IF (gu8_SystemState = DRIVE_SYS AND DO_q_BatteryDischargeMain_DO = TRUE) THEN
	IF (gq_Gear_Drive_Rq = TRUE AND gq_BrakeSwitch = TRUE) AND gr_VehicleSpeed_kmph > -1 THEN
		gq_Gear_Neutral			:=	FALSE;
		gq_Gear_Drive			:=	TRUE;
		gq_Gear_DriveCrawl		:=	FALSE;
		gq_Gear_Reverse			:=	FALSE;
		gq_Gear_ReverseCrawl	:=	FALSE; (*Select Drive*)
	ELSIF (gq_Gear_Neutral_Rq = TRUE AND gq_BrakeSwitch = TRUE) AND (gr_VehicleSpeed_kmph <1 AND gr_VehicleSpeed_kmph >-1) THEN
		gq_Gear_Neutral			:=	TRUE;
		gq_Gear_Drive			:=	FALSE;
		gq_Gear_DriveCrawl		:=	FALSE;
		gq_Gear_Reverse			:=	FALSE;
		gq_Gear_ReverseCrawl	:=	FALSE; (*Select Neutral*)
	ELSIF (gq_Gear_Reverse_Rq = TRUE AND gq_BrakeSwitch = TRUE) AND gr_VehicleSpeed_kmph < 1 THEN
		gq_Gear_Neutral			:=	FALSE;
		gq_Gear_Drive			:=	FALSE;
		gq_Gear_DriveCrawl		:=	FALSE;
		gq_Gear_Reverse			:=	TRUE;
		gq_Gear_ReverseCrawl	:=	FALSE; (*Select Reverse*)
	ELSIF (DI_q_DirectionSwitch_DriveCrawl_DI = TRUE AND gq_BrakeSwitch = TRUE) THEN
		gq_Gear_Neutral			:=	FALSE;
		gq_Gear_Drive			:=	FALSE;
		gq_Gear_DriveCrawl		:=	TRUE;
		gq_Gear_Reverse			:=	FALSE;
		gq_Gear_ReverseCrawl	:=	FALSE; (*Select Drive Crawl*)
	(*ELSIF (DI_q_DirectionSwitch_ReverseCrawl_DI = TRUE AND gq_BrakeSwitch = TRUE) THEN
		gq_Gear_Neutral			:=	FALSE;
		gq_Gear_Drive			:=	FALSE;
		gq_Gear_DriveCrawl		:=	FALSE;
		gq_Gear_Reverse			:=	FALSE;
		gq_Gear_ReverseCrawl	:=	TRUE; (*Select Reverse Crawl*)*)
	END_IF
ELSIF (gu8_SystemState <> DRIVE_SYS) THEN
	gq_Gear_Neutral			:=	TRUE;
	gq_Gear_Drive			:=	FALSE;
	gq_Gear_DriveCrawl		:=	FALSE;
	gq_Gear_Reverse			:=	FALSE;
	gq_Gear_ReverseCrawl	:=	FALSE; (*Gear selection = Neutral*)
ELSE
	gq_Gear_Neutral			:=	TRUE;
	gq_Gear_Drive			:=	FALSE;
	gq_Gear_DriveCrawl		:=	FALSE;
	gq_Gear_Reverse			:=	FALSE;
	gq_Gear_ReverseCrawl	:=	FALSE; (*Neutral*)
END_IF

gq_ReverseLights	:=	gq_Gear_Reverse;

END_PROGRAM

// Application/UserCode/BMS/OrionBMS/Orion_Control
PROGRAM Orion_Control
VAR
	OrionPause_Timer	:	TON;
	hton_DisconnectionPause_Timer	:	TON;
END_VAR

(*Program to control the BMS during operation*)
(*Setting battery mode*)
IF (gu8_SystemState = DRIVE_SYS) THEN
	(*Have an initial short pause after contactors have closed before changing into discharge mode*)
	OrionPause_Timer(IN := TRUE, PT := T#20mS);
	IF (OrionPause_Timer.Q = TRUE) THEN
		(*Set discharge output*)
		DO_q_DrivetrainKL15C_DO	:=	FALSE;
		DO_q_DrivetrainKL15D_DO	:=	TRUE;
		(*Request on CAN the BMS into operational mode*)
		gu8_BMS1_MPO_1_State	:=	1;
		gu8_BMS1_MPO_2_State	:=	1; (* This does F_ALL *)
		gu8_BMS2_MPO_1_State	:=	1;
		gu8_BMS2_MPO_2_State	:=	1;
		
		
	END_IF
	hton_DisconnectionPause_Timer(IN := FALSE, PT := T#0MS);
ELSIF (gu8_SystemState = PLUGIN_SYS) THEN
	(*Have an initial short pause after contactors have closed before changing into charge mode*)
	OrionPause_Timer(IN := TRUE, PT := T#20MS);
	IF (OrionPause_Timer.Q = TRUE) THEN
		(*Set outputs for charge mode*)
		DO_q_DrivetrainKL15C_DO	:=	TRUE;
		DO_q_DrivetrainKL15D_DO	:=	FALSE;
		(*Request on CAN the BMS into operational mode*)
		gu8_BMS1_MPO_1_State	:=	0;
		gu8_BMS1_MPO_2_State	:=	0;
		gu8_BMS2_MPO_1_State	:=	0;
		gu8_BMS2_MPO_2_State	:=	0;
	END_IF
	hton_DisconnectionPause_Timer(IN := FALSE, PT := T#0MS);
ELSIF (DO_q_BatteryDischargeMain_DO = FALSE AND DO_q_Battery1ChargeMain_DO = FALSE AND DO_q_Battery2ChargeMain_DO = FALSE AND
		DO_q_BatteryDischargePrecharge_DO = FALSE AND DO_q_Battery1ChargePrecharge_DO = FALSE AND DO_q_Battery2ChargePrecharge_DO = FALSE) THEN
	(*Only perform disconnect of batteries when all contactors are opened to prevent them from damaging their own contactors Explain ??MAT *)
	hton_DisconnectionPause_Timer(IN := TRUE, PT := T#100MS);
	IF (hton_DisconnectionPause_Timer.Q = TRUE) THEN
		DO_q_DrivetrainKL15C_DO	:=	FALSE;
		DO_q_DrivetrainKL15D_DO	:=	FALSE;
		(*Request the BMS inactive*)
		gu8_BMS1_MPO_1_State	:=	0;
		gu8_BMS1_MPO_2_State	:=	0;
		gu8_BMS2_MPO_1_State	:=	0;
		gu8_BMS2_MPO_2_State	:=	0;
			
	END_IF
	OrionPause_Timer(IN := FALSE, PT := t#0ms);
END_IF
IF qq_BMS1_PB_DTC_Reset THEN
	gu8_BMS1_MPO_3_State :=1;
	ELSE gu8_BMS1_MPO_3_State :=0;
END_IF
IF qq_BMS2_PB_DTC_Reset THEN
	gu8_BMS2_MPO_3_State :=1;
	ELSE gu8_BMS2_MPO_3_State :=0;
END_IF

END_PROGRAM

// Application/UserCode/MCU/MCU_Control
PROGRAM MCU_Control
VAR
	hs8_Direction	:	SINT	:=	0;
	hton_Mileometer	:	TON;
	hq_SetInitialDistance	:	BOOL	:=	FALSE;
	hton_TorqueRqRamp	:	TON;
	hr_TorqueRampTime	:	REAL;
	hr_TorqueRampTotal	:	REAL;
	hr_MCU_TorquePreRamp	:	REAL;
	hf_TorqueRamp			:	Ramp_Linear;
	
	TORQUE_RQ_CF	:	REAL	:=	0.3; (*In case any conversion factors need to be applied to the value being sent*)
	hr_MULTIPLIER_CALC	: REAL	:= 0;
	WINDUPSPEED			: USINT := 10;
	
	hr_SpeedLimit_KP	:	REAL	:=	10;
	hr_SpeedLimit_KI	:	REAL	:=	10;
	hfb_SpeedLimit_PID	:	PID;
	hr_MaximumTorqueLimit : REAL;
	hr_TARGETMAXSPEED : REAL := 77;
	hr_IntegralCounter : ARRAY [0..49] OF REAL;
	Counter : USINT := 0;
	hr_IntegralSum : REAL := 0;
	Cycle : USINT;
END_VAR
VAR CONSTANT
	INITIALISATION	:	USINT	:=	0;
	STANDBY			:	USINT	:=	1;
	STARTUP			:	USINT	:=	2;
	TEARDOWN		:	USINT	:=	3;
	OPERATIONAL		:	USINT	:=	4;
	FAILURE			:	USINT	:=	5;
	CLOSEDOWN		:	USINT	:=	6;
	READYTOSHUTDOWN	:	USINT	:=	7;
	WAITFORCOOLING	:	USINT	:=	8;
	
	SHUTDOWN_RQ		:	USINT	:=	2;
	OPERATIONAL_RQ	:	USINT	:=	1;
	STANDBY_RQ		:	USINT	:=	0;
	
	TORQUE_MODE		:	USINT	:=	1;
	SPEED_MODE		:	USINT	:=	2;
	
	
	
	EV_MODE			:	USINT	:=	3;
	NEU_NOTORQUE	:	USINT	:=	0;

END_VAR

IF (DI_q_VehicleKL15_DI = TRUE) THEN
	hton_Mileometer(IN := TRUE, PT := T#60S);
	IF (gu16_MCU_MaxMotorSpeed_Rx = 0) THEN
		gu8_MCU_VMUPollMCU_Multiplex	:=	MAXMOTORSPEED;
	ELSIF (gu16_MCU_MaxMotorTorque_Rx = 0) THEN
		gu8_MCU_VMUPollMCU_Multiplex	:=	MAXMOTORTORQUE;
	ELSIF (hton_Mileometer.Q = TRUE) THEN
		hton_Mileometer(IN := FALSE, PT := T#0S);
		gu8_MCU_VMUPollMCU_Multiplex	:=	TOTALMOTORROTATION;
	ELSE
		gu8_MCU_VMUPollMCU_Multiplex	:=	8; (*Not applicable value so will not incorrectly request any data*)
	END_IF
END_IF

(*Must be in discharge mode and precharge complete before command out of standby (Need to set ignition at the start always)*)
IF (gu8_SystemState = DRIVE_SYS AND DOS_q_BatteryDischargeMain_DO = TRUE(* AND gr_MCU_TractionTorqueAvailable > 0*)) THEN
	IF ((gu8_MCU_State = STANDBY) AND gq_Gear_Neutral = TRUE) THEN
		gu8_MCU_OperationRequest	:=	OPERATIONAL_RQ;
		gu8_MCU_OperationalMode_Tx	:=	NEU_NOTORQUE;
	ELSIF (gu8_MCU_State = OPERATIONAL) THEN
		gu8_MCU_OperationRequest	:=	OPERATIONAL_RQ;
		gu8_MCU_OperationalMode_Tx	:=	EV_MODE;
	END_IF
ELSIF (gu8_SystemState <> DRIVE_SYS) THEN
	IF (gu8_MCU_State = OPERATIONAL AND gq_Gear_Neutral = TRUE) THEN
		gu8_MCU_OperationRequest	:=	SHUTDOWN_RQ;
		gu8_MCU_OperationalMode_Tx	:=	NEU_NOTORQUE;
	ELSIF (gu8_MCU_State = OPERATIONAL AND gq_Gear_Neutral = FALSE) THEN
		gu8_MCU_OperationRequest	:=	OPERATIONAL_RQ;
		gu8_MCU_OperationalMode_Tx	:=	NEU_NOTORQUE;
		(*Rq Neutral*)
	ELSE
		gu8_MCU_OperationRequest	:=	STANDBY_RQ;
		gu8_MCU_OperationalMode_Tx	:=	NEU_NOTORQUE;
	END_IF
ELSE
	gu8_MCU_OperationRequest	:=	STANDBY_RQ;
	gu8_MCU_OperationalMode_Tx	:=	NEU_NOTORQUE;
END_IF

(*These values should be set by the BMS*)
gu16_MCU_MaxChargeCurrent		:=	REAL_TO_UINT(gr_BMS_CCL);
gu16_MCU_MaxDischargeCurrent	:=	REAL_TO_UINT(gr_BMS_DCL);
gu16_MCU_MaxBatteryVoltage		:=	gu16_BMS_Maximum_Pack_Voltage;
gu16_MCU_MinBatteryVoltage		:=	gu16_BMS_MinimumPackVoltage;
gu8_MCU_CommandMode				:=	TORQUE_MODE;
gu8_MCU_ReferenceCommandMode	:=	TORQUE_MODE;
gr_MCU_MaxMotorSpeed_PreCF		:=	gr_MCU_MaxMotorSpeed; (*This may need to be set for safety*)

IF (gq_Gear_Drive = TRUE OR gq_Gear_DriveCrawl = TRUE) THEN
	hs8_Direction	:=	1;
	gq_MCU_SpeedCommandStatus		:=	FALSE;
	gq_MCU_TorqueCommandStatus		:=	FALSE;
ELSIF (gq_Gear_Reverse = TRUE OR gq_Gear_ReverseCrawl = TRUE) THEN
	hs8_Direction	:=	-1;
	gq_MCU_SpeedCommandStatus		:=	FALSE;
	gq_MCU_TorqueCommandStatus		:=	FALSE;
ELSE
	hs8_Direction	:=	0;
	gq_MCU_SpeedCommandStatus		:=	TRUE;
	gq_MCU_TorqueCommandStatus		:=	TRUE;
END_IF

hr_MULTIPLIER_CALC := gr_VehicleSpeed_kmph / WINDUPSPEED;
TORQUE_RQ_CF := LIMIT(1(*0.3*), hr_MULTIPLIER_CALC, 1);

Driveability();
IF (gu8_MCU_State = OPERATIONAL AND hs8_Direction <> 0 (*Not in neutral*) AND gq_ABSActive = FALSE AND gq_MCU_CutOff_LowCellV = FALSE AND gq_BodySteps = FALSE) THEN
	IF (gq_ABS_TorqueDisable = TRUE) THEN
		hton_TorqueRqRamp(IN := FALSE, PT := T#0S);
		gr_MCU_TorqueCommand_PreCF			:=	0;
	ELSIF (gq_ZeroTorqueRq = TRUE) THEN
		hton_TorqueRqRamp(IN := FALSE, PT := T#0S);
		IF (gq_RegenActive = TRUE) THEN
			gr_MCU_TorqueCommand_PreCF	:=	(*gr_MCU_MaxMotorTorque*)gr_MCU_RegenTorqueAvailable * gr_RegenSOCMultiplier * gr_RegenMultiplierRq * gr_RegenSpeedDegrading * gr_RegenIntroCF * (hs8_Direction * (-1)) * LIMIT(0, (gr_TorqueReIntro / gr_TorqueReIntroMax), 1);(**)
		ELSIF (gq_RegenActive = FALSE) THEN
			gr_MCU_TorqueCommand_PreCF			:=	gr_AccelPedal_Perc * TORQUE_RQ_CF * hs8_Direction * (*gr_MCU_MaxMotorTorque*)gr_MCU_TractionTorqueAvailable * LIMIT(0, (gr_TorqueReIntro / gr_TorqueReIntroMax), 1);
		END_IF
	ELSIF (gq_ABS_TorqueDisable = FALSE AND gq_ZeroTorqueRq = FALSE) THEN
		IF (gq_RegenActive = TRUE) THEN
			hton_TorqueRqRamp(IN := FALSE, PT := T#0S);
			gr_MCU_TorqueCommand_PreCF	:=	(*gr_MCU_MaxMotorTorque*)gr_MCU_RegenTorqueAvailable * gr_RegenSOCMultiplier * gr_RegenMultiplierRq * gr_RegenSpeedDegrading * gr_RegenIntroCF * (hs8_Direction * (-1));(**)
		ELSIF (gq_RegenActive = FALSE) THEN	
			hr_MCU_TorquePreRamp	:=	gr_AccelPedal_Perc * TORQUE_RQ_CF * hs8_Direction * (*gr_MCU_MaxMotorTorque*)gr_MCU_TractionTorqueAvailable;
			gr_MCU_TorqueCommand_PreCF	:=	hr_MCU_TorquePreRamp;
		END_IF
	END_IF
	//*DO_q_DrivetrainCoolingFan_DO		:=	TRUE;
ELSE
	gr_MCU_TorqueCommand_PreCF			:=	0 * TORQUE_RQ_CF * (*gr_MCU_MaxMotorTorque*)gr_MCU_TractionTorqueAvailable;
	//*DO_q_DrivetrainCoolingFan_DO		:=	FALSE;
	hton_TorqueRqRamp(IN := FALSE, PT := T#0S);
END_IF

IF (gu8_BMS_SOC > 10) THEN
	IF (gu8_ChassisType <> CHASSIS_IVECO) THEN
		hr_TARGETMAXSPEED := SpeedOTG;
	ELSIF (gu8_ChassisType = CHASSIS_IVECO) THEN
		hr_TARGETMAXSPEED := 55;
	END_IF
ELSE
	IF (gu8_ChassisType <> CHASSIS_IVECO) THEN
		hr_TARGETMAXSPEED := SpeedOTG1;
	ELSIF (gu8_ChassisType = CHASSIS_IVECO) THEN
		hr_TARGETMAXSPEED := 24;
	END_IF
END_IF

IF (gr_VehicleSpeed_kmph > hr_TARGETMAXSPEED) THEN
	hr_MaximumTorqueLimit := 0;
ELSE
	hr_IntegralCounter[Counter] := LIMIT(0, (hr_TARGETMAXSPEED - gr_VehicleSpeed_kmph), hr_TARGETMAXSPEED);
	IF (Counter > 49) THEN
		Counter := 0;
	ELSE
		Counter := Counter + 1;
	END_IF
	hr_IntegralSum := 0;
	FOR Cycle := 0 TO 49 DO
		hr_IntegralSum := hr_IntegralSum + hr_IntegralCounter[Cycle];
	END_FOR
	hr_MaximumTorqueLimit := MAX(((hr_TARGETMAXSPEED - gr_VehicleSpeed_kmph) * hr_SpeedLimit_KP + hr_IntegralSum * hr_SpeedLimit_KI), 0);
END_IF


gr_MCU_SpeedCommand_PreCF			:=	0;

gr_MCU_TorqueCommand_PreCF_Limited	:=	LIMIT(-3500, gr_MCU_TorqueCommand_PreCF, hr_MaximumTorqueLimit);
gr_MCU_ReferenceTorqueCommand_PreCF	:=	LIMIT(-3500, gr_MCU_TorqueCommand_PreCF, hr_MaximumTorqueLimit);
gr_MCU_ReferenceSpeedCommand_PreCF	:=	gr_MCU_SpeedCommand_PreCF;

(*Don't think I need to set these but will keep them here as a reminder and just in case they do need setting*)
gq_MCU_MaxDiscahrgeCurrentStatus	:=	FALSE;
gq_MCU_MaxBatteryVoltageStatus		:=	FALSE;
gq_MCU_MinBatteryVoltageStatus		:=	FALSE;
gq_MCU_MaxChargeCurrentStatus		:=	FALSE;

gr_VehicleSpeed_kmph	:=	f_SpeedCalc(gr_MotorSpeed_IN := gr_MCU_MotorSpeed, gu16_GearRatio_IN := gu16_GearRatio_PreCF,
										gu16_DyfRatio_IN := gu16_DyfRatio_PreCF, gu16_TireWidth_IN := gu16_TireWidth_mm,
										gu8_TireProfile_IN := gu8_TireProfile_Perc, gu16_WheelDiameter_IN := gu16_WheelDiameter_PreCF);

gr_VehicleAllTimeDistance	:=	f_DistanceCalc(gr_MotorRotation_IN := gr_MCU_TotalMotorRotation, gu16_GearRatio_IN := gu16_GearRatio_PreCF,
										gu16_DyfRatio_IN := gu16_DyfRatio_PreCF, gu16_TireWidth_IN := gu16_TireWidth_mm,
										gu8_TireProfile_IN := gu8_TireProfile_Perc, gu16_WheelDiameter_IN := gu16_WheelDiameter_PreCF);

IF (hq_SetInitialDistance = FALSE AND gr_MCU_TotalMotorRotation <> 0) THEN
	gr_VehicleInitialTripDistance	:=	gr_VehicleAllTimeDistance;
	hq_SetInitialDistance			:=	TRUE;
END_IF

gr_VehicleTripDistance	:=	gr_VehicleAllTimeDistance - gr_VehicleInitialTripDistance;

END_PROGRAM

// Application/UserCode/MCU/Driveability
PROGRAM Driveability
VAR
	hq_RegenAvailable	:	BOOL;
	hton_RegenHysteresis	:	TON;
	hr_DriveSpeed	:	REAL;
	hr_FrontSpeed	:	REAL;
	hr_LeftWheels_Speed	:	REAL;
	hr_RightWheels_Speed	:	REAL;
	hr_TractionSpdDiff	:	REAL;
	hr_StabilitySpdDiff	:	REAL;
	
	(*Traction and Stability Dennis and Iveco*)
	TRACTIONLOSS_RELSPEED	:	REAL	:=	300; (*Temporarily set high until time to configure these to the correct value*)
	STABLOSS_RELSPEED		:	REAL	:=	3; (*Temporarily set high until time to configure these to the correct value*)
	(*Bob traction and stability values*)
	TRACTIONLOSS_SPEED	:	UINT	:=	3500;
	STABLOSS_SPEED		:	UINT	:=	1000;
	
	REGEN_CUTOFF_SPEED	:	USINT	:=	5;
	REGEN_WINDDOWNABOVECUTOFF_SPEED	:	USINT	:=	25;
	hton_RegenStartTimer : TON;
	// This ideally should be set to 100ms
	htime_RegenIntro : TIME := T#100MS;
	
	// WAS 0.7 ON BRAKE
	DENNIS_ADJUSTABLE_REGEN	:	REAL	:=	0.4 (*0.4*);
	
	hr_StabilityRelativeDifference : REAL;
	hu8_StabRampSpeed	:	USINT	:=	30;
	hr_STABLOSS_HIGHSPD	:	REAL	:=	2.5;
	hr_StabIncreaseMultiplier	:	REAL	:=	3;
	hr_STABLOSS_HIGHSPD_IVECO	:	REAL	:=	1.5;
	hr_StabIncreaseMultiplier_IVECO	:	REAL	:=	2;
	
	hr_RegenTest	:	REAL	:=	1; (*Use this value in place of the constants for regen multiplier to allow changes to be made by forcing on the fly*)
	
	SecretTractionOff: BOOL;
	hton_Overspeed_Regen: TON;
END_VAR
VAR_INPUT
	Dennis_Regen_Selector: BYTE := 0;
END_VAR


(*ABS*)
IF (CAN3_Rx.Mode_Button AND CAN3_Rx.Down_Button) = TRUE THEN
	SecretTractionOff :=	TRUE;
END_IF

IF (CAN3_Rx.Mode_Button AND CAN3_Rx.Up_Button) = TRUE THEN
	SecretTractionOff := 	FALSE;
END_IF

IF (gq_ABSActive = TRUE) THEN
	gq_ABS_TorqueDisable	:=	TRUE;
ELSIF (gq_ABSActive = FALSE AND gr_AccelPedal_Perc > 0.03(*3%*)) THEN
	gq_ABS_TorqueDisable	:=	FALSE;
END_IF

IF (gq_Frosty_NoWheelSpeedSensors = TRUE) THEN
	hr_STABLOSS_HIGHSPD_IVECO	:=	10; (*Set so that Stability loss detection does not prevent drive*)
END_IF

IF (gu8_ChassisType = CHASSIS_IVECO AND gq_StabTracDisable_Rx = FALSE) THEN
	(*Traction Control*)
	gr_RearAxle_RelativeSpeed_kph	:= (gr_EBC2_KB_RearRight1RelSpd + gr_EBC2_KB_RearLeft1RelSpd) / 2;
	IF (ABS(gr_RearAxle_RelativeSpeed_kph) > TRACTIONLOSS_RELSPEED(*Change this value to be whatever the speed difference needs to be to trigger can be decimal*)) THEN
		gu8_TractionLoss	:=	1(*TRUE*);
	ELSE
		gu8_TractionLoss	:=	0(*FALSE*);
	END_IF

	(*Stability*)
	IF (gr_VehicleSpeed_kmph > hu8_StabRampSpeed) THEN
		STABLOSS_RELSPEED := hr_STABLOSS_HIGHSPD_IVECO;
	ELSE
		STABLOSS_RELSPEED := hr_STABLOSS_HIGHSPD_IVECO + ((hu8_StabRampSpeed - ABS(gr_VehicleSpeed_kmph)) * hr_StabIncreaseMultiplier_IVECO / hu8_StabRampSpeed);
	END_IF
	
	gr_LeftWheels_RelativeSpeed_kph		:=	(gr_EBC2_KB_FrontLeftRelSpd + gr_EBC2_KB_RearLeft1RelSpd) / 2;
	gr_RightWheels_RelativeSpeed_kph	:=	(gr_EBC2_KB_FrontRightRelSpd + gr_EBC2_KB_RearRight1RelSpd) / 2;
	IF (ABS(gr_LeftWheels_RelativeSpeed_kph) > STABLOSS_RELSPEED OR ABS(gr_RightWheels_RelativeSpeed_kph) > STABLOSS_RELSPEED) THEN (*Can equally use decimal numbers here if needed*)
		gu8_StabilityLoss	:=	1(*TRUE*);
	ELSE
		gu8_StabilityLoss	:=	0(*FALSE*);
	END_IF
ELSIF (gu8_ChassisType = CHASSIS_BOB OR gu8_ChassisType = CHASSIS_ESTARGLIDER) AND (gq_StabTracDisable_Rx = FALSE AND SecretTractionOff = FALSE) THEN // OR should be AND
	(*Traction Control*)
	hr_DriveSpeed	:= (gu16_Bob_RightDrive_CAN + gu16_Bob_LeftDrive_CAN) / 2;
	hr_FrontSpeed	:= (gu16_Bob_RightFront_CAN + gu16_Bob_LeftFront_CAN) / 2;
	hr_TractionSpdDiff	:=	ABS(hr_DriveSpeed - hr_FrontSpeed);
	IF (hr_TractionSpdDiff > TRACTIONLOSS_SPEED(*Change this value to be whatever the speed difference needs to be to trigger can be decimal*)) THEN
		gu8_TractionLoss	:=	1(*TRUE*);
	ELSE
		gu8_TractionLoss	:=	0(*FALSE*);
	END_IF
	(*Stability*)
	hr_LeftWheels_Speed		:=	(gu16_Bob_LeftFront_CAN + gu16_Bob_LeftDrive_CAN) / 2;
	hr_RightWheels_Speed	:=	(gu16_Bob_RightFront_CAN + gu16_Bob_RightDrive_CAN) / 2;
	hr_StabilitySpdDiff		:=	ABS(hr_LeftWheels_Speed - hr_RightWheels_Speed);
	IF (hr_StabilitySpdDiff > STABLOSS_SPEED) THEN (*Can equally use decimal numbers here if needed*)
		gu8_StabilityLoss	:=	1(*TRUE*);
	ELSE
		gu8_StabilityLoss	:=	0(*FALSE*);
	END_IF
ELSIF (gu8_ChassisType = CHASSIS_DENNIS AND (gq_StabTracDisable_Rx = FALSE AND SecretTractionOFF = FALSE)) THEN
	(*Traction Control*)
	(*gr_RearAxle_RelativeSpeed_kph	:= (gr_EBC2_KB_RearRight1RelSpd + gr_EBC2_KB_RearLeft1RelSpd) / 2;
	IF (ABS(gr_RearAxle_RelativeSpeed_kph) > TRACTIONLOSS_RELSPEED(*Change this value to be whatever the speed difference needs to be to trigger can be decimal*)) THEN
		gu8_TractionLoss	:=	1(*TRUE*);
	ELSE
		gu8_TractionLoss	:=	0(*FALSE*);
	END_IF*)
	(*Stability*)
	IF (gr_VehicleSpeed_kmph > hu8_StabRampSpeed) THEN
		STABLOSS_RELSPEED := hr_STABLOSS_HIGHSPD;
	ELSE
		STABLOSS_RELSPEED := hr_STABLOSS_HIGHSPD + ((hu8_StabRampSpeed - ABS(gr_VehicleSpeed_kmph)) * hr_StabIncreaseMultiplier / hu8_StabRampSpeed);
	END_IF
	
	gr_LeftWheels_RelativeSpeed_kph		:=	(gr_EBC2_KB_FrontLeftRelSpd + gr_EBC2_KB_RearLeft1RelSpd) / 2;
	gr_RightWheels_RelativeSpeed_kph	:=	(gr_EBC2_KB_FrontRightRelSpd + gr_EBC2_KB_RearRight1RelSpd) / 2;
	hr_StabilityRelativeDifference	:=	ABS(gr_LeftWheels_RelativeSpeed_kph - gr_RightWheels_RelativeSpeed_kph);
	IF (*(ABS(gr_LeftWheels_RelativeSpeed_kph) > STABLOSS_RELSPEED OR ABS(gr_RightWheels_RelativeSpeed_kph) > STABLOSS_RELSPEED)*)
		(hr_StabilityRelativeDifference > STABLOSS_RELSPEED) THEN (*Can equally use decimal numbers here if needed*)
		gu8_StabilityLoss	:=	1(*TRUE*);
	ELSE
		gu8_StabilityLoss	:=	0(*FALSE*);
	END_IF
	gu8_TractionLoss	:=	gu8_EBC1_ASREngineControlActive;
	(*gu8_StabilityLoss	:=	gu8_EBC1_ASRBrakeControlActive;*)
ELSIF (gq_StabTracDisable_Rx = TRUE) THEN
	gu8_TractionLoss	:=	0(*FALSE*);
	gu8_StabilityLoss	:=	0(*FALSE*);
END_IF


(*Zero torque and Recovery*)
IF (gu8_TractionLoss = 1 OR gu8_StabilityLoss = 1 (* REAMED by IAIN 121021 OR Sevcon2_Control.NO_OIL*)) THEN
	gq_ZeroTorqueRq	:=	TRUE;
	gton_TorqueReIntro_Timer(IN := FALSE, PT := T#0MS);
ELSE
	gton_TorqueReIntro_Timer(IN := TRUE, PT := T#2000MS);
END_IF
IF (gton_TorqueReIntro_Timer.Q = TRUE) THEN
	gq_ZeroTorqueRq	:=	FALSE;
END_IF
gr_TorqueReIntro	:=	TIME_TO_REAL(gton_TorqueReIntro_Timer.ET);
gr_TorqueReIntroMax	:=	TIME_TO_REAL(T#2000MS);

(*Regen*)
(*Selectable regen setting needed*)
IF (gu8_BMS_SOC < 90) THEN
	gr_RegenSOCMultiplier	:=	1;
ELSIF (gu8_BMS_SOC >= 90 AND gu8_BMS_SOC < 95) THEN
	gr_RegenSOCMultiplier	:=	0.5;
ELSE
	gr_RegenSOCMultiplier	:=	0;
END_IF


IF (gr_VehicleSpeed_kmph > REGEN_CUTOFF_SPEED) THEN
	hton_RegenHysteresis(IN := TRUE, PT := T#1000MS); // bring down to T#1s? Was t#5s
ELSE
	hton_RegenHysteresis(IN := FALSE, PT := T#0S);
END_IF
hq_RegenAvailable	:=	hton_RegenHysteresis.Q;

hton_Overspeed_Regen (IN:= gr_VehicleSpeed_kmph > 55, PT:= T#5S);
IF ((gr_AccelPedal_Perc < 0.01 OR (gr_VehicleSpeed_kmph > 55 AND hton_Overspeed_Regen.Q)) AND hq_RegenAvailable = TRUE) THEN //OR gr_VehicleSpeed_kmph > 56 added
	gq_RegenActive	:=	TRUE;
	gr_RegenSpeedDegrading	:=	LIMIT(0, (gr_VehicleSpeed_kmph - REGEN_CUTOFF_SPEED), REGEN_WINDDOWNABOVECUTOFF_SPEED) / REGEN_WINDDOWNABOVECUTOFF_SPEED;
	IF gr_VehicleSpeed_kmph > 55 THEN
	DENNIS_ADJUSTABLE_REGEN := 1.2;
	END_IF
//////////////	

//DENNIS with BRAKE
	IF (gu8_ChassisType = CHASSIS_DENNIS AND gq_BrakeSwitch = TRUE) THEN
		DENNIS_ADJUSTABLE_REGEN := 1.2;
		gr_RegenMultiplierRq	:=	DENNIS_ADJUSTABLE_REGEN;
		hton_RegenStartTimer(IN := TRUE, PT := htime_RegenIntro);
		gr_RegenIntroCF := LIMIT(0, (TIME_TO_REAL(hton_RegenStartTimer.ET) / TIME_TO_REAL(hton_RegenStartTimer.PT)), 1);
	END_IF
//DENNIS without BRAKE	
	IF (gu8_ChassisType = CHASSIS_DENNIS AND gq_BrakeSwitch = FALSE) THEN
		gr_RegenMultiplierRq	:=	DENNIS_ADJUSTABLE_REGEN(*40%*);
		hton_RegenStartTimer(IN := TRUE, PT := htime_RegenIntro);
		gr_RegenIntroCF := LIMIT(0, (TIME_TO_REAL(hton_RegenStartTimer.ET) / TIME_TO_REAL(hton_RegenStartTimer.PT)), 1);
		
		IF Dennis_Regen.RegenCounterValue = 0 THEN 
			DENNIS_ADJUSTABLE_REGEN := 0;
		END_IF
		IF Dennis_Regen.RegenCounterValue = 1 THEN
			DENNIS_ADJUSTABLE_REGEN := 0.6;
		END_IF
		IF Dennis_Regen.RegenCounterValue = 2 THEN
			DENNIS_ADJUSTABLE_REGEN := 0.8;
		END_IF
		IF Dennis_Regen.RegenCounterValue = 3 THEN
			DENNIS_ADJUSTABLE_REGEN := 1;
		END_IF
		IF Dennis_Regen.RegenCounterValue = 4 THEN
			DENNIS_ADJUSTABLE_REGEN := 1.2;
		END_IF	
//////////////		

ELSIF (gq_BrakeSwitch = TRUE AND gu8_ChassisType <> CHASSIS_DENNIS) THEN
		IF (gu8_RegenSelector = 0) THEN
			gr_RegenMultiplierRq	:=	0.7(*40%*);
			hton_RegenStartTimer(IN := TRUE, PT := htime_RegenIntro);
			gr_RegenIntroCF := LIMIT(0, (TIME_TO_REAL(hton_RegenStartTimer.ET) / TIME_TO_REAL(hton_RegenStartTimer.PT)), 1);
		ELSIF (gu8_RegenSelector = 1) THEN
			gr_RegenMultiplierRq	:=	0.7(*40%*);
			hton_RegenStartTimer(IN := TRUE, PT := htime_RegenIntro);
			gr_RegenIntroCF := LIMIT(0, (TIME_TO_REAL(hton_RegenStartTimer.ET) / TIME_TO_REAL(hton_RegenStartTimer.PT)), 1);
		ELSIF (gu8_RegenSelector = 2) THEN
			gr_RegenMultiplierRq	:=	0.7(*60%*);
			hton_RegenStartTimer(IN := TRUE, PT := htime_RegenIntro);
			gr_RegenIntroCF := LIMIT(0, (TIME_TO_REAL(hton_RegenStartTimer.ET) / TIME_TO_REAL(hton_RegenStartTimer.PT)), 1);
		END_IF
	ELSIF (gq_BrakeSwitch = FALSE AND gu8_ChassisType <> CHASSIS_DENNIS) THEN
		IF (gu8_RegenSelector = 0) THEN
			gr_RegenMultiplierRq	:=	0(*0%*);
			hton_RegenStartTimer(IN := FALSE, PT := T#0MS);
			gr_RegenIntroCF := 0;
		ELSIF (gu8_RegenSelector = 1) THEN
			gr_RegenMultiplierRq	:=	0.6(*0.4(*40%*)*);
			hton_RegenStartTimer(IN := TRUE, PT := htime_RegenIntro);
			gr_RegenIntroCF := LIMIT(0, (TIME_TO_REAL(hton_RegenStartTimer.ET) / TIME_TO_REAL(hton_RegenStartTimer.PT)), 1);
		ELSIF (gu8_RegenSelector = 2) THEN
			gr_RegenMultiplierRq	:=	1(*0.6(*60%*)*);
			hton_RegenStartTimer(IN := TRUE, PT := htime_RegenIntro);
			gr_RegenIntroCF := LIMIT(0, (TIME_TO_REAL(hton_RegenStartTimer.ET) / TIME_TO_REAL(hton_RegenStartTimer.PT)), 1);
		END_IF
	END_IF
ELSE
	gq_RegenActive	:=	FALSE;
	gr_RegenMultiplierRq	:=	0;
	hton_RegenStartTimer(IN := FALSE, PT := T#0MS);
	gr_RegenIntroCF := 0;
END_IF
(*Also need battery SOC as multiplier <90 x1, 90<X<95 x0.5, >95 x0*)





(*Creep / Hill hold*)

END_PROGRAM

// Application/UserCode/Sevcon_Compressor/Sevcon2_Control
PROGRAM Sevcon2_Control
VAR
	hton_WindUpTorque_Timer	:	TON;
	hton_AirPressureExceeded_Timer	:	TON;
	htof_AirpressureRelief_Timer	:	TOF;
	hq_AirCompressorEnable	:	BOOL;
	hton_AirPressureDelayTimer	:	TON;
	
	hq_AirReliefValveOff : BOOL;
	
	
	hton_Compressor_Oil_Switch: TON;
	Low_Oil: BOOL;
	NO_OIL: BOOL;
	Oil_Temp_Setpoint: BYTE := 30;
	Oil_Level_Warning: BOOL;
	Compressor_Temp_Warning: BOOL;
	Comp_Motor_Temp_SP_Warning: INT := 100; //LM change from 55
	Comp_Motor_Temp_SP_Fault: INT := 120;  //LM change from 65
	Compressor_Temp_Fault: BOOL;
	Air_Temp_SP_Warning: INT := 100;
	Air_Temp_SP_Fault: INT := 120;
	Air_Temp_Warning: BOOL;
	Air_Temp_Fault: BOOL;
	BlowOffTime: TIME := T#1S;
	AirSuspensionPressure: REAL := 14.9;
	APRTimerET: TIME := t#0.5s;
	AirPressureReliefTime: TIME := t#1s;
	hton_Compressor_Run_Timer: TON;
	CRT_Trigger: BOOL;
	CRT_Time: TIME := t#60s;
	Run_on_Brake_Pressure: REAL := 9.5;
	CRT_Timer: TON;
	PVCT: TON;
	PVCT_Time: TIME := T#60s;
END_VAR
VAR CONSTANT
	(*Statuswords*)
	NOTREADY_STAT				:	USINT	:=	1;
	SHUTDOWN_STAT				:	USINT	:=	2;
	PRECHARGE_STAT				:	USINT	:=	4;
	ENERGISED_STAT				:	USINT	:=	7;
	ENABLED_STAT				:	USINT	:=	8;
	FAULTREACTIONACTIVE_STAT	:	USINT	:=	11;
	FAULTOFF_STAT				:	USINT	:=	13;
	ACTIVESHORT_STAT			:	USINT	:=	14;
	(*Commandwords*)
	NOCOMMAND_COMM		:	USINT	:=	0;
	ENERGISE_COMM		:	USINT	:=	3;
	ENABLED_COMM		:	USINT	:=	5;
	SHUTDOWN_COMM		:	USINT	:=	6;
	FAULTRESET_COMM		:	USINT	:=	9;
	ACTIVESHORT_COMM	:	USINT	:=	10;
	
	(*LOWAIRPRESSURE		:	REAL	:=	7.2; (*Need to define what the low air pressure value that is reported is*)
	HIGHAIRPRESSURE		:	REAL	:=	10;
	LOWAIRPRESSURE_BOB		:	REAL	:=	10; (*Need to define what the low air pressure value that is reported is*)
	HIGHAIRPRESSURE_BOB		:	REAL	:=	12.2(*Glider*) (*12.3 for Bob*);*)
	
	
	TORQUE_RQ			:	USINT	:=	200;
	REVERSE_SPD_LIMIT	:	INT		:=	-500;
	MAX_DISCHARGE		:	USINT	:=	50;
	MAX_CHARGE			:	SINT	:=	-50;
	TRACTION_LIMIT		:	USINT	:=	100;
END_VAR


(**)
(*Check for Comms fault*)
IF (gu8_SystemState = DRIVE_SYS AND DOS_q_BatteryDischargeMain_DO = TRUE) THEN
	IF (gu8_Sevcon2_InverterStatus = FAULTOFF_STAT OR gu8_Sevcon2_InverterStatus = ACTIVESHORT_STAT) THEN
		gu16_Sevcon2_Controlword	:=	FAULTRESET_COMM;
	ELSIF (gu8_Sevcon2_InverterStatus = NOTREADY_STAT OR gu8_Sevcon2_InverterStatus = SHUTDOWN_STAT) THEN
		gu16_Sevcon2_Controlword	:=	ENERGISE_COMM;
	ELSIF (gu8_Sevcon2_InverterStatus = PRECHARGE_STAT) THEN
		gu16_Sevcon2_Controlword	:=	ENERGISE_COMM;
	ELSIF (gu8_Sevcon2_InverterStatus = ENERGISED_STAT) THEN
		gu16_Sevcon2_Controlword	:=	ENABLED_COMM;
	ELSIF (gu8_Sevcon2_InverterStatus = ENABLED_STAT) THEN
		gu16_Sevcon2_Controlword	:=	ENABLED_COMM; (*Need a way to switch off*)
	ELSE
		gu16_Sevcon2_Controlword	:=	NOCOMMAND_COMM;
	END_IF
ELSE
	gu16_Sevcon2_Controlword	:=	SHUTDOWN_COMM;
END_IF

CRT_Timer (IN:= NOT hq_AirCompressorEnable, PT := CRT_Time); //Active when compressor hasnt run
hton_AirPressureDelayTimer(IN := TRUE, PT := T#2000MS);
PVCT (IN :=  hq_AirCompressorEnable, PT := PVCT_Time); // Compressor run-on timer

IF (hton_AirPressureDelayTimer.Q = TRUE) THEN
	IF (gq_APU_Installed = FALSE) THEN
		IF 	//(gr_J1939_AirSuspensionSupplyPress > gr_HighAirPressure_CutOff OR
			(gr_J1939_ServiceBrakeAirPressCircuit1 > gr_HighAirPressure_CutOff OR
			gr_J1939_ServiceBrakeAirPressCircuit2 > gr_HighAirPressure_CutOff) THEN
			hton_AirPressureExceeded_Timer(IN := TRUE, PT := BlowOffTime);
		ELSE
			hton_AirPressureExceeded_Timer(IN := FALSE, PT := T#1S); //changed from 0 to 2s to increase hysteresis
		END_IF
		IF (gu8_SystemState = DRIVE_SYS AND DOS_q_BatteryDischargeMain_DO = TRUE AND
			NO_OIL = FALSE AND Compressor_Temp_Fault = FALSE) (*AND gq_Bob_AirCompressorStatus_CAN = TRUE)*) THEN
			IF  (gr_VehicleSpeed_kmph > 5 AND (gr_J1939_ServiceBrakeAirPressCircuit1 < Run_on_Brake_Pressure)) OR // added to increase duty cycle
				
				//(PVCT.Q = FALSE AND CRT_Timer.Q = TRUE AND gr_VehicleSpeed_kmph > 2) OR // runs compressor for a time period
				
				((gr_J1939_AirSuspensionSupplyPress < gr_LowAirPressure_Intro OR
				gr_J1939_ServiceBrakeAirPressCircuit1 < gr_LowAirPressure_Intro OR
				gr_J1939_ServiceBrakeAirPressCircuit2 < gr_LowAirPressure_Intro) AND
				gq_DriveMode_CutOff_LowCellV = FALSE) THEN
					gu16_Sevcon2_SpeedLimitForward	:=	2600; (*Controlling the speed through the limits*)
					hq_AirCompressorEnable	:=	TRUE;
			ELSIF ((hton_AirPressureExceeded_Timer.Q = TRUE) OR (gr_VehicleSpeed_kmph > 5 AND (gr_J1939_ServiceBrakeAirPressCircuit1 > Run_on_Brake_Pressure))) THEN
				//(PVCT.Q = TRUE AND CRT_Timer.Q = FALSE AND gr_VehicleSpeed_kmph < 2) THEN // added to increase duty cycle
				gu16_Sevcon2_SpeedLimitForward	:=	0;
				hq_AirCompressorEnable	:=	FALSE;
			END_IF
		ELSE
			gu16_Sevcon2_SpeedLimitForward	:=	0;
			hq_AirCompressorEnable	:=	FALSE;
		END_IF
	
	(*For Bob possibly use
	(*gq_Bob_AirCompressorStatus_CAN = FALSE AND hq_AirReliefValveOff = TRUE)*)
	See below for how it was implemented*)
		
	(*This is needed for when the compressor is being controlled by the APU not yet*)
	ELSE
		(*IF (gr_J1939_AirSuspensionSupplyPress > HIGHAIRPRESSURE_BOB AND
			(gr_J1939_ServiceBrakeAirPressCircuit1 > HIGHAIRPRESSURE_BOB AND
			gr_J1939_ServiceBrakeAirPressCircuit2 > HIGHAIRPRESSURE_BOB))				
			(*gq_Bob_AirCompressorStatus_CAN = FALSE AND hq_AirReliefValveOff = TRUE)*) THEN
			hton_AirPressureExceeded_Timer(IN := TRUE, PT := T#1000MS);
		ELSE
			hton_AirPressureExceeded_Timer(IN := FALSE, PT := T#0MS);
		END_IF*)
		IF (gu8_SystemState = DRIVE_SYS AND DOS_q_BatteryDischargeMain_DO = TRUE AND
			NO_OIL = FALSE AND Compressor_Temp_Fault = FALSE AND gq_Bob_AirCompressorStatus_CAN = TRUE) THEN
			IF (gq_Merc_AirComp_Rq = TRUE AND gq_DriveMode_CutOff_LowCellV = FALSE) OR (htof_AirpressureRelief_Timer.ET > APRTimerET) THEN
					gu16_Sevcon2_SpeedLimitForward	:=	2600; (*Controlling the speed through the limits*)
					hq_AirCompressorEnable	:=	TRUE;
			ELSE(*ELSIF (hton_AirPressureExceeded_Timer.Q = TRUE) THEN*)
				gu16_Sevcon2_SpeedLimitForward	:=	0;
				hq_AirCompressorEnable	:=	FALSE;
			END_IF
		ELSE
			gu16_Sevcon2_SpeedLimitForward	:=	0;
			hq_AirCompressorEnable	:=	FALSE;
		END_IF
		(*hq_AirReliefValveOff := gq_Bob_AirCompressorStatus_CAN;*)
	END_IF
END_IF
(*gq_Merc_AirComp_Enabled	:=	hq_AirCompressorEnable;*)


htof_AirpressureRelief_Timer(IN := gq_Merc_AirComp_Rq, PT := AirPressureReliefTime);
IF htof_AirpressureRelief_Timer.Q THEN
	hq_AirCompressorEnable	:=	TRUE;
	(*(hq_AirCompressorEnable = TRUE AND gs16_Sevcon2_SpeedMeasured < 1000 )) THEN*)
	gu16_Sevcon2_SpeedLimitForward	:=	2600; (*Controlling the speed through the limits*)
	hq_AirCompressorEnable	:=	TRUE;
ELSE
		;
END_IF


(*All these are constants to be sent out to the Sevcon unit and do not need changing during operation*)
IF (gu8_Sevcon2_InverterStatus = ENABLED_STAT) THEN
	hton_WindUpTorque_Timer(IN := TRUE, PT := T#5000MS);
	gr_Sevcon2_TorqueRq						:=	TORQUE_RQ * (TIME_TO_REAL(hton_WindUpTorque_Timer.ET) / 5000);
ELSE
	hton_WindUpTorque_Timer(IN := FALSE, PT := T#0MS);
	gr_Sevcon2_TorqueRq						:=	0;
END_IF
	
gr_Sevcon2_DCLink_VoltageTarget			:=	0; (*Not needed as not being used as a generator*)
gs16_Sevcon2_SpeedLimitReverse			:=	REVERSE_SPD_LIMIT;
gu16_Sevcon2_DCLink_ImaxDischarge		:=	MAX_DISCHARGE;
gs16_Sevcon2_DCLink_ImaxRecharge		:=	MAX_CHARGE;
gr_Sevcon2_TorqueTractionLimit			:=	TRACTION_LIMIT;
gr_Sevcon2_TorqueRegenLimit				:=	0;

gu8_Sevcon2_CSCommand1					:=	0;
gu8_Sevcon2_CSCommand2					:=	0;
gu8_Sevcon2_CSCurrentLimits				:=	0;
(*Counters to run every cycle and increment so the Sevcons know the VMU is still running*)
IF (gu8_Sevcon2_SEQCommand1 < 255) THEN
	gu8_Sevcon2_SEQCommand1			:=	gu8_Sevcon2_SEQCommand1 + 1;
ELSE
	gu8_Sevcon2_SEQCommand1			:=	0;
END_IF
IF (gu8_Sevcon2_SEQCommand2 < 255) THEN
	gu8_Sevcon2_SEQCommand2			:=	gu8_Sevcon2_SEQCommand2 + 1;
ELSE
	gu8_Sevcon2_SEQCommand2			:=	0;
END_IF
IF (gu8_Sevcon2_SEQCurrentLimits < 255) THEN
	gu8_Sevcon2_SEQCurrentLimits	:=	gu8_Sevcon2_SEQCurrentLimits + 1;
ELSE
	gu8_Sevcon2_SEQCurrentLimits	:=	0;
END_IF
(**************************************************************)
hton_Compressor_Oil_Switch(IN:= Low_Oil, PT:= T#2M);
IF Sevcon2_Rx.Compressor_Oil_Switch < 1 (*Rimmed AND gs16_Sevcon2_MotorTemp < Oil_Temp_Setpoint *) AND  gs16_Sevcon2_SpeedMeasured <2000 THEN
	Low_Oil := FALSE; (*changed due to poor switching*)
ELSE
	Low_Oil := FALSE;
END_IF

IF hton_Compressor_Oil_Switch.Q THEN
	NO_OIL := FALSE;
ELSE
	NO_OIL := FALSE;
END_IF

IF hton_Compressor_Oil_Switch.ET > T#30S THEN
	Oil_Level_Warning := TRUE;
ELSE
	Oil_Level_Warning := FALSE;
END_IF

IF gs16_Sevcon2_MotorTemp > Comp_Motor_Temp_SP_Warning THEN
	Compressor_Temp_Warning	:= TRUE;
ELSE
	Compressor_Temp_Warning	:= FALSE;
END_IF

IF	gs16_Sevcon2_MotorTemp > Comp_Motor_Temp_SP_Fault THEN
	Compressor_Temp_Fault := TRUE;
ELSE
	Compressor_Temp_fault := FALSE;
END_IF

IF	Sevcon2_Rx.Compressor_Temperature > Air_Temp_SP_Warning THEN
	Air_Temp_Warning := TRUE;
ELSE
	Air_Temp_Warning := FALSE;
END_IF

IF	Sevcon2_Rx.Compressor_Temperature > Air_Temp_SP_Fault THEN
	Air_Temp_Fault := TRUE;
ELSE
	Air_Temp_Fault := FALSE;
END_IF

END_PROGRAM

// Application/UserCode/MCU/f_SpeedCalc
FUNCTION f_SpeedCalc : REAL
VAR_INPUT
	gr_MotorSpeed_IN		:	REAL;
	gu16_GearRatio_IN		:	UINT;
	gu16_DyfRatio_IN		:	UINT;
	gu16_TireWidth_IN		:	UINT;
	gu8_TireProfile_IN		:	USINT;
	gu16_WheelDiameter_IN	:	UINT;
END_VAR
VAR
	hr_SidewallWidth_m	:	REAL;
	hr_TotalWheelDiameter_m	:	REAL;
	hr_WheelCircumfrence_km	:	REAL;
	hr_RevsPerKm			:	REAL;
	
	hr_GearRatio				:	REAL;
	hr_DyfRatio					:	REAL;
	hr_WheelDiameter_inch		:	REAL;
	hr_WheelDiameter_m			:	REAL;
END_VAR
VAR CONSTANT
	PI	:	REAL	:=	3.14159;
	INCH_TO_METER_CF	:	REAL	:=	0.0254;
	MILLI_TO_METER		:	UINT	:=	1000;
END_VAR


hr_GearRatio				:=	gu16_GearRatio_IN / 1000;
hr_DyfRatio					:=	gu16_DyfRatio_IN / 1000;
hr_WheelDiameter_inch		:=	gu16_WheelDiameter_IN / 10;

hr_WheelDiameter_m			:=	hr_WheelDiameter_inch * INCH_TO_METER_CF;
hr_SidewallWidth_m			:=	gu16_TireWidth_mm * (gu8_TireProfile_Perc / 100) / MILLI_TO_METER;
hr_TotalWheelDiameter_m		:=	hr_WheelDiameter_m + hr_SidewallWidth_m;

hr_WheelCircumfrence_km		:=	(hr_TotalWheelDiameter_m * PI) / 1000;
hr_RevsPerKm				:=	1 / hr_WheelCircumfrence_km;

f_SpeedCalc	:=	gr_MotorSpeed_IN / hr_GearRatio / hr_DyfRatio / hr_RevsPerKm * 60;

END_FUNCTION

// Application/UserCode/MCU/f_DistanceCalc
FUNCTION f_DistanceCalc : REAL
VAR_INPUT
	gr_MotorRotation_IN		:	REAL;
	gu16_GearRatio_IN		:	UINT;
	gu16_DyfRatio_IN		:	UINT;
	gu16_TireWidth_IN		:	UINT;
	gu8_TireProfile_IN		:	USINT;
	gu16_WheelDiameter_IN	:	UINT;
END_VAR
VAR
	hr_SidewallWidth_m	:	REAL;
	hr_TotalWheelDiameter_m	:	REAL;
	hr_WheelCircumfrence_km	:	REAL;
	hr_RevsPerKm			:	REAL;
	
	hr_GearRatio				:	REAL;
	hr_DyfRatio					:	REAL;
	hr_WheelDiameter_inch		:	REAL;
	hr_WheelDiameter_m			:	REAL;
END_VAR
VAR CONSTANT
	PI	:	REAL	:=	3.14159;
	INCH_TO_METER_CF	:	REAL	:=	0.0254;
	MILLI_TO_METER		:	UINT	:=	1000;
END_VAR


hr_GearRatio				:=	gu16_GearRatio_IN / 1000;
hr_DyfRatio					:=	gu16_DyfRatio_IN / 1000;
hr_WheelDiameter_inch		:=	gu16_WheelDiameter_IN / 10;

hr_WheelDiameter_m			:=	hr_WheelDiameter_inch * INCH_TO_METER_CF;
hr_SidewallWidth_m			:=	gu16_TireWidth_mm * (gu8_TireProfile_Perc / 100) / MILLI_TO_METER;
hr_TotalWheelDiameter_m		:=	hr_WheelDiameter_m + hr_SidewallWidth_m;

hr_WheelCircumfrence_km		:=	(hr_TotalWheelDiameter_m * PI) / 1000;
hr_RevsPerKm				:=	1 / hr_WheelCircumfrence_km;

f_DistanceCalc	:=	gr_MotorRotation_IN / hr_GearRatio / hr_DyfRatio / hr_RevsPerKm;

END_FUNCTION

// Application/UserCode/BELDCDC/BELDCDC_Control
PROGRAM BELDCDC_Control
VAR
	hton_DelayTimer	:	TON;
END_VAR

(*Setting the digital outputs to the DCDC*)

IF (DOS_q_BatteryDischargeMain_DO = TRUE AND gu8_SystemState = DRIVE_SYS) THEN
	(*Once the main contactor is connected wait 5 seconds then set the ouputs high*)
	hton_DelayTimer(IN := TRUE, PT := T#5S);
	DO_q_DrivetrainDCDCInhibit_DO	:=	hton_DelayTimer.Q;
	DO_q_DashboardDCDCStatus_DO		:=	hton_DelayTimer.Q;
ELSIF (DO_q_Battery1ChargeMain_DO = TRUE OR DO_q_Battery2ChargeMain_DO = TRUE) THEN
	(*Switch off outputs when in charge*)
	hton_DelayTimer(IN := FALSE, PT := T#0S);
	DO_q_DrivetrainDCDCInhibit_DO	:=	FALSE;
	DO_q_DashboardDCDCStatus_DO		:=	FALSE;
	(*This is included for future so that the DCDC can be brought in during charge but is not possible with current electrical setup*)
ELSE
	(*Any other state switch outputs off*)
	hton_DelayTimer(IN := FALSE, PT := T#0S);
	DO_q_DrivetrainDCDCInhibit_DO	:=	FALSE;
	DO_q_DashboardDCDCStatus_DO		:=	FALSE;
END_IF

END_PROGRAM

// Application/UserCode/Sevcon_PSP/Sevcon_Steer_Control
PROGRAM Sevcon_Steer_Control
VAR
	hton_WindUpTorque_Timer	:	TON;
	hq_PowerSteering_Enable	:	BOOL;
	hton_HandbrakeOffTimer	:	TON;
	hr_SteeringSpeed		:	REAL;
	hton_PowerSteeringOff	:	TON;
	Steering_Speed_Setpoint: INT := 2200; //changed from 2000
END_VAR
VAR CONSTANT
	(*Statuswords*)
	NOTREADY_STAT				:	USINT	:=	1;
	SHUTDOWN_STAT				:	USINT	:=	2;
	PRECHARGE_STAT				:	USINT	:=	4;
	ENERGISED_STAT				:	USINT	:=	7;
	ENABLED_STAT				:	USINT	:=	8;
	FAULTREACTIONACTIVE_STAT	:	USINT	:=	11;
	FAULTOFF_STAT				:	USINT	:=	13;
	ACTIVESHORT_STAT			:	USINT	:=	14;
	(*Commandwords*)
	NOCOMMAND_COMM		:	USINT	:=	0;
	ENERGISE_COMM		:	USINT	:=	3;
	ENABLED_COMM		:	USINT	:=	5;
	SHUTDOWN_COMM		:	USINT	:=	6;
	FAULTRESET_COMM		:	USINT	:=	9;
	ACTIVESHORT_COMM	:	USINT	:=	10;
	
	TORQUE_RQ			:	USINT	:=	200;
	REVERSE_SPD_LIMIT	:	INT		:=	-500;
	MAX_DISCHARGE		:	USINT	:=	50;
	MAX_CHARGE			:	SINT	:=	-50;
	TRACTION_LIMIT		:	USINT	:=	100;
	
	CANBUS_OFF			:	INT	:=	21256;
END_VAR


(**)
(*Check for Comms fault*)
IF (gu8_SystemState = DRIVE_SYS AND DOS_q_BatteryDischargeMain_DO = TRUE) THEN
	DO_q_DrievtrainPowerSteering_DO	:=	TRUE;
	IF (gu8_Sevcon1_InverterStatus = FAULTOFF_STAT OR gu8_Sevcon1_InverterStatus = ACTIVESHORT_STAT) THEN
		gu16_Sevcon1_Controlword	:=	FAULTRESET_COMM;
	ELSIF (gu8_Sevcon1_InverterStatus = NOTREADY_STAT OR gu8_Sevcon1_InverterStatus = SHUTDOWN_STAT) THEN
		gu16_Sevcon1_Controlword	:=	ENERGISE_COMM;
	ELSIF (gu8_Sevcon1_InverterStatus = PRECHARGE_STAT) THEN
		gu16_Sevcon1_Controlword	:=	ENERGISE_COMM;
	ELSIF (gu8_Sevcon1_InverterStatus = ENERGISED_STAT) THEN
		gu16_Sevcon1_Controlword	:=	ENABLED_COMM;
	ELSIF (gu8_Sevcon1_InverterStatus = ENABLED_STAT) THEN
		gu16_Sevcon1_Controlword	:=	ENABLED_COMM;
	ELSE
		gu16_Sevcon1_Controlword	:=	NOCOMMAND_COMM;
	END_IF
ELSE
	DO_q_DrievtrainPowerSteering_DO	:=	FALSE;
	gu16_Sevcon1_Controlword	:=	SHUTDOWN_COMM;
END_IF

hton_HandbrakeOffTimer(IN := HMI_Rx.gq_Dennis_Handbrake, PT := T#10MS); //Time changed from 30s to 10ms

(*This could be changed to link to the current speed of the vehicle in which case the different gear ratios and wheel diameter will be needed here to calculate*)
IF ((HMI_Rx.gq_Dennis_Handbrake = FALSE OR NOT gq_Gear_Neutral) AND gu8_SystemState = DRIVE_SYS) THEN //TEST FIRST THEN REMOVE THIS COMMENT OR NOT gq_Gear_Neutral
	hq_PowerSteering_Enable	:=	TRUE;
	hr_SteeringSpeed		:=	MAX(REAL_TO_INT(Steering_Speed_Setpoint - (ABS(gr_VehicleSpeed_kmph) * 10)), 0) (*Ensure the speed limit is never set negative*);
	gu16_Sevcon1_SpeedLimitForward	:=	REAL_TO_UINT(LIMIT(200, hr_SteeringSpeed, Steering_Speed_Setpoint)); (*Controlling the speed through the limits*)
	hton_PowerSteeringOff(IN := FALSE, PT := T#0S);
ELSIF ((hton_HandbrakeOffTimer.Q = TRUE AND ABS(gr_VehicleSpeed_kmph) < 3) AND gu8_SystemState = DRIVE_SYS) THEN //AND before DRIVE_SYS changed from OR
	hq_PowerSteering_Enable	:=	FALSE;
	hton_PowerSteeringOff(IN := TRUE, PT := T#10MS);
	
	IF (hton_PowerSteeringOff.Q = TRUE) THEN
		gu16_Sevcon1_SpeedLimitForward	:=	200; //instead of shutting off reduce speed to a minimum
	ELSE
		gu16_Sevcon1_SpeedLimitForward	:=	650;
	END_IF
	
END_IF


(*All these are constants to be sent out to the Sevcon unit and do not need changing during operation*)
IF (gu8_Sevcon1_InverterStatus = ENABLED_STAT) THEN
	hton_WindUpTorque_Timer(IN := TRUE, PT := T#5000MS);
	gr_Sevcon1_TorqueRq						:=	TORQUE_RQ * (TIME_TO_REAL(hton_WindUpTorque_Timer.ET) / 5000);
ELSE
	hton_WindUpTorque_Timer(IN := FALSE, PT := T#0MS);
	gr_Sevcon1_TorqueRq						:=	0;
END_IF

gr_Sevcon1_DCLink_VoltageTarget			:=	0; (*Not needed as not being used as a generator*)
gs16_Sevcon1_SpeedLimitReverse			:=	REVERSE_SPD_LIMIT;
gu16_Sevcon1_DCLink_ImaxDischarge		:=	MAX_DISCHARGE;
gs16_Sevcon1_DCLink_ImaxRecharge		:=	MAX_CHARGE;
gr_Sevcon1_TorqueTractionLimit			:=	TRACTION_LIMIT;
gr_Sevcon1_TorqueRegenLimit				:=	0;

gu8_Sevcon1_CSCommand1					:=	0;
gu8_Sevcon1_CSCommand2					:=	0;
gu8_Sevcon1_CSCurrentLimits				:=	0;

(*Counters to run every cycle and increment so the Sevcons know the VMU is still running*)
IF (gu8_Sevcon1_SEQCommand1 < 255) THEN
	gu8_Sevcon1_SEQCommand1			:=	gu8_Sevcon1_SEQCommand1 + 1;
ELSE
	gu8_Sevcon1_SEQCommand1			:=	0;
END_IF
IF (gu8_Sevcon1_SEQCommand2 < 255) THEN
	gu8_Sevcon1_SEQCommand2			:=	gu8_Sevcon1_SEQCommand2 + 1;
ELSE
	gu8_Sevcon1_SEQCommand2			:=	0;
END_IF
IF (gu8_Sevcon1_SEQCurrentLimits < 255) THEN
	gu8_Sevcon1_SEQCurrentLimits	:=	gu8_Sevcon1_SEQCurrentLimits + 1;
ELSE
	gu8_Sevcon1_SEQCurrentLimits	:=	0;
END_IF

(*Backup Pump*)
IF (hq_PowerSteering_Enable = TRUE AND gs16_Sevcon1_FaultCode = CANBUS_OFF) THEN (* Matt, does something else need ORed*)
	DO_q_BackupPump_DO	:=	TRUE;
	(*Fault state will set from the sevcon error*)
ELSE
	DO_q_BackupPump_DO	:=	FALSE;
END_IF

END_PROGRAM

// Application/UserCode/CAN4/Heater/Heater_Control
PROGRAM Heater_Control
VAR
	HEATER_VALUE_Low	:	USINT	:=	20;
	HEATER_VALUE_Med	:	USINT	:=	40;
	HEATER_VALUE_High	:	USINT	:=	80;
	// Temperature request 110(dec) - 50 deg C = 60degC
	HEATER_TEMP_60C: USINT := 110;
	// Temperature request 100(dec) - 50 deg C = 50degC
	HEATER_TEMP_50C: USINT := 100;
	// Temperature request 90(dec) - 50 deg C = 40degC
	HEATER_TEMP_40C: USINT := 90;
END_VAR


IF	gq_HMI_Heater_Enable = FALSE THEN
	gu8_Heater_Perc		:=	0;
	gu8_Heater_Temp_Tx	:=	0;
	gq_HeaterPumpEnable	:=	FALSE;
ELSE
	gq_HeaterPumpEnable	:=	TRUE;
	gq_Heater_EnableBit := TRUE;
END_IF

IF (gq_HMI_Heater_Enable = TRUE) AND (gq_HMI_Heater_Low = TRUE) AND (gu8_systemstate = 1) THEN
		gu8_Heater_Perc		:=	HEATER_VALUE_High;
		gu8_Heater_Temp_Tx	:=	HEATER_TEMP_40C;
	ELSIF (gq_HMI_Heater_Enable	= TRUE) AND (gq_HMI_Heater_Med = TRUE) THEN
		gu8_Heater_Perc		:=	HEATER_VALUE_High;
		gu8_Heater_Temp_Tx	:=	HEATER_TEMP_50C; 
	ELSIF (gq_HMI_Heater_Enable	=	TRUE) AND (gq_HMI_Heater_Hi = TRUE) THEN
		gu8_Heater_Perc		:=	HEATER_VALUE_High;
		gu8_Heater_Temp_Tx	:=	HEATER_TEMP_60C;
	END_IF

END_PROGRAM

// Application/UserCode/ePTO/ePTO_Control
PROGRAM ePTO_Control
VAR
	hu16_TORQUEREFHIGH	: UINT	:=	90; (*%*)
	hu16_TORQUEREFLOW	: UINT	:=	0;	(*%*)
	hu16_SPEEDTARGET	: UINT	:=	1150; (*RPM*)
	hs16_FAN_On_Temp	: INT	:=	60; (*degC*)
	hs16_FAN_Off_Temp	: INT	:=	50;	(*degC*)
	
	hton_CANOpen_Start_Timer	:	TON;
	hton_CANOpen_StartCommand_OtherAddress_Timer	:	TON;
	hu16_IdleSpeedTarget: UINT := 250;
	BinLiftTimer: TON;
	BinLiftTime: TIME := t#3s;
END_VAR


gu16_TrqHi	:=	(hu16_TORQUEREFHIGH * 50) + 5000;
gu16_TrqLo	:=	(hu16_TORQUEREFLOW * 50) + 5000;
gu8_Asym_Limits	:=	16#20;

IF ((gs16_InverterTemp > hs16_FAN_On_Temp) OR (gs16_MotorTemp > hs16_FAN_On_Temp)) THEN
	gu8_DIGITAL1	:=	16#80;
ELSIF ((gs16_InverterTemp < hs16_FAN_Off_Temp) AND (gs16_MotorTemp < hs16_FAN_Off_Temp)) THEN
	gu8_DIGITAL1	:=	16#0;
END_IF

BinLiftTimer (IN:= (gq_Gear_Drive = TRUE OR gq_Gear_Reverse = TRUE), PT:= BinLiftTime);

IF (DOS_q_BatteryDischargeMain_DO = TRUE) THEN
	(*Activate Motor*)
	IF (gu8_ePTO_ActivationByte <> 0) OR (BinLiftTimer.Q = FALSE AND gq_Gear_Neutral = FALSE) THEN
		gu16_Skai_SpeedTarget	:=	hu16_SPEEDTARGET + 32768;
		gq_ePTO_Activate	:=	TRUE;
	ELSE
		gu16_Skai_SpeedTarget	:=	hu16_IdleSpeedTarget + 32768; (*added to allow permanent running of ePTO*)
		gq_ePTO_Activate	:=	TRUE(*FALSE*);
	END_IF
ELSE
	gu16_Skai_SpeedTarget	:=	32768; (*Offset so value is actually 0*)
	gq_ePTO_Activate	:=	FALSE;
END_IF


(*CANOpen*)
hton_CANOpen_Start_Timer(IN := TRUE, PT := T#5S);
hton_CANOpen_StartCommand_OtherAddress_Timer(IN := hton_CANOpen_Start_Timer.Q, PT := T#1S);
IF (hton_CANOpen_Start_Timer.Q = TRUE) THEN
	gu8_CANOpen_Command	:=	16#01;
	gu8_CANOpen_NodeAddress	:=	16#7A;
ELSIF (hton_CANOpen_StartCommand_OtherAddress_Timer.Q = TRUE) THEN
	gu8_CANOpen_Command	:=	16#01;
	gu8_CANOpen_NodeAddress	:=	16#7B;
ELSE
	gu8_CANOpen_Command	:=	16#81;
	gu8_CANOpen_NodeAddress	:=	16#7A;
END_IF

gq_ePTO_FanEnable	:=	gq_ePTO_Activate;

END_PROGRAM

// Application/UserCode/Main Program/Project_Infomation
PROGRAM Project_Infomation


VAR
	Project_Name: STRING(255);
	Description: STRING(255);
	Profile: STRING(255);
	Last_Change: STRING(255);
	ver: STRING(255);
	Major: BYTE;
	Minor: BYTE;
	patch: BYTE;
END_VAR

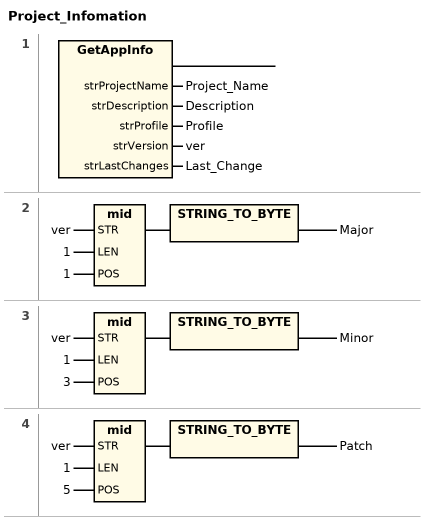
// NETWORK 1
GetAppInfo(strProjectName => Project_Name, strDescription => Description, strProfile => Profile, strVersion => ver, strLastChanges => Last_Change);

// NETWORK 2
Major := STRING_TO_BYTE(mid(STR := ver, LEN := 1, POS := 1));

// NETWORK 3
Minor := STRING_TO_BYTE(mid(STR := ver, LEN := 1, POS := 3));

// NETWORK 4
Patch := STRING_TO_BYTE(mid(STR := ver, LEN := 1, POS := 5));

END_PROGRAM

// Application/UserCode/Main Program/GetAppInfo
FUNCTION GetAppInfo : BOOL
(*'******************************************************************************
'* This Function gets the application information.
'*
'* Function requires the system library CmpApp
'* 
'*******************************************************************************
*)
VAR_OUTPUT
   strProjectName: STRING(255);
   strDescription: STRING(255);
   strProfile: STRING(255);
   strVersion: STRING(255);
   strLastChanges: STRING(255);
END_VAR
VAR
   tResult: DWORD;
   tFirstApp: POINTER TO APPLICATION;
   pAppInfo: POINTER TO APPLICATION_INFO;
   pString : POINTER TO STRING;
END_VAR

tFirstApp := AppGetFirstApp(pResult := tResult);
IF tFirstApp <> 0 THEN
   pAppInfo :=AppGetApplicationInfo(tFirstApp, tResult);
   strProjectName :=pAppInfo^.pstProjectName^;
   strDescription:=pAppInfo^.pstDescription^;
   strProfile:=pAppInfo^.pstProfile^;
   strVersion:=pAppInfo^.pstVersion^;
   strLastChanges:=DT_TO_STRING(pAppInfo^.dtLastChanges);
END_IF

END_FUNCTION

// Application/UserCode/BMS/OrionBMS/OrionBMS_Tx
PROGRAM OrionBMS_Tx
VAR
	ht_OrionBMS1_State_Tx	:	EPEC_CANVXD.Msg;
	ht_OrionBMS2_State_Tx	:	EPEC_CANVXD.Msg;
	hton_MessageSend_Timer	:	TON;
END_VAR

(*Transmit control of both BMS*)

(*Setup output message structure with ID, Data and Length*)
ht_OrionBMS1_State_Tx.ID	:=	16#023;
ht_OrionBMS1_State_Tx.Data[0]	:=	gu8_BMS1_MPO_1_State;
ht_OrionBMS1_State_Tx.Data[1]	:=	gu8_BMS1_MPO_2_State;
ht_OrionBMS1_State_Tx.Data[2]	:=	gu8_BMS1_MPO_3_State;
ht_OrionBMS1_State_Tx.Data[3]	:=	gu8_BMS1_MPO_4_State;
ht_OrionBMS1_State_Tx.Data[4]	:=	gu8_BMS1_MPE_State;
ht_OrionBMS1_State_Tx.Data[5]	:=	0;
ht_OrionBMS1_State_Tx.Data[6]	:=	0;
ht_OrionBMS1_State_Tx.Data[7]	:=	0;
ht_OrionBMS1_State_Tx.Len	:=	8;

(*Setup output message structure with ID, Data and Length*)
ht_OrionBMS2_State_Tx.ID	:=	16#023;
ht_OrionBMS2_State_Tx.Data[0]	:=	gu8_BMS2_MPO_1_State;
ht_OrionBMS2_State_Tx.Data[1]	:=	gu8_BMS2_MPO_2_State;
ht_OrionBMS2_State_Tx.Data[2]	:=	gu8_BMS2_MPO_3_State;
ht_OrionBMS2_State_Tx.Data[3]	:=	gu8_BMS2_MPO_4_State;
ht_OrionBMS2_State_Tx.Data[4]	:=	gu8_BMS2_MPE_State;
ht_OrionBMS2_State_Tx.Data[5]	:=	0;
ht_OrionBMS2_State_Tx.Data[6]	:=	0;
ht_OrionBMS2_State_Tx.Data[7]	:=	0;
ht_OrionBMS2_State_Tx.Len	:=	8;

(*Same message needed for both BMS so structure for BMS1 saved across into BMS2   NOW SEPERATE!!*)
(*ht_OrionBMS2_State_Tx	:=	ht_OrionBMS1_State_Tx;*)

(*Message broadcast timer and actual structure send on CANbus*)
hton_MessageSend_Timer(IN := NOT(hton_MessageSend_Timer.Q), PT := T#100MS);
IF (hton_MessageSend_Timer.Q = TRUE) THEN
	G_CAN2_Channel.SendMessage(i_pMSG:=ADR(ht_OrionBMS1_State_Tx));
	G_CAN3_Channel.SendMessage(i_pMSG:=ADR(ht_OrionBMS2_State_Tx));
END_IF

END_PROGRAM

// Application/UserCode/Sevcon_PSP/Sevcon_Steer_Tx
PROGRAM Sevcon_Steer_Tx
VAR
	ht_TorqueDemand1_Tx			:	EPEC_CANVXD.Msg;
	ht_TorqueDemand2_Tx			:	EPEC_CANVXD.Msg;
	ht_BatteryDemand_Tx			:	EPEC_CANVXD.Msg;
	ht_DirectIControlDemand_Tx	:	EPEC_CANVXD.Msg;
	hton_SendTimer				:	TON;
END_VAR

Sevcon_Steer_TxConversion();

ht_TorqueDemand1_Tx.ID		:=	16#191071FA OR EPEC_CANVXD.MASK_29BIT;
ht_TorqueDemand1_Tx.Data[0]	:=	UINT_TO_USINT(gu16_Sevcon1_TorqueRq_Tx);
ht_TorqueDemand1_Tx.Data[1]	:=	UINT_TO_USINT(SHR(gu16_Sevcon1_TorqueRq_Tx, 8));
ht_TorqueDemand1_Tx.Data[2]	:=	UINT_TO_USINT(gu16_Sevcon1_Controlword);
ht_TorqueDemand1_Tx.Data[3]	:=	UINT_TO_USINT(SHR(gu16_Sevcon1_Controlword, 8));
ht_TorqueDemand1_Tx.Data[4]	:=	UINT_TO_USINT(gu16_Sevcon1_TorqueTractionLimit_Tx);
ht_TorqueDemand1_Tx.Data[5]	:=	UINT_TO_USINT(SHR(gu16_Sevcon1_TorqueTractionLimit_Tx, 8));
ht_TorqueDemand1_Tx.Data[6]	:=	gu8_Sevcon1_SEQCommand1;
ht_TorqueDemand1_Tx.Data[7]	:=	gu8_Sevcon1_CSCommand1;
ht_TorqueDemand1_Tx.Len	:=	8;

ht_TorqueDemand2_Tx.ID		:=	16#191171FA OR EPEC_CANVXD.MASK_29BIT;
ht_TorqueDemand2_Tx.Data[0]	:=	UINT_TO_USINT(gu16_Sevcon1_TorqueRegenLimit_Tx);
ht_TorqueDemand2_Tx.Data[1]	:=	UINT_TO_USINT(SHR(gu16_Sevcon1_TorqueRegenLimit_Tx, 8));
ht_TorqueDemand2_Tx.Data[2]	:=	UINT_TO_USINT(gu16_Sevcon1_SpeedLimitForward);
ht_TorqueDemand2_Tx.Data[3]	:=	UINT_TO_USINT(SHR(gu16_Sevcon1_SpeedLimitForward, 8));
ht_TorqueDemand2_Tx.Data[4]	:=	INT_TO_USINT(gs16_Sevcon1_SpeedLimitReverse);
ht_TorqueDemand2_Tx.Data[5]	:=	INT_TO_USINT(SHR(gs16_Sevcon1_SpeedLimitReverse, 8));
ht_TorqueDemand2_Tx.Data[6]	:=	gu8_Sevcon1_SEQCommand2;
ht_TorqueDemand2_Tx.Data[7]	:=	gu8_Sevcon1_CSCommand2;
ht_TorqueDemand2_Tx.Len		:=	8;

ht_BatteryDemand_Tx.ID		:=	16#191271FA OR EPEC_CANVXD.MASK_29BIT;
ht_BatteryDemand_Tx.Data[0]	:=	UINT_TO_USINT(gu16_Sevcon1_DCLink_ImaxDischarge);
ht_BatteryDemand_Tx.Data[1]	:=	UINT_TO_USINT(SHR(gu16_Sevcon1_DCLink_ImaxDischarge, 8));
ht_BatteryDemand_Tx.Data[2]	:=	INT_TO_USINT(gs16_Sevcon1_DCLink_ImaxRecharge);
ht_BatteryDemand_Tx.Data[3]	:=	INT_TO_USINT(SHR(gs16_Sevcon1_DCLink_ImaxRecharge, 8));
ht_BatteryDemand_Tx.Data[4]	:=	UINT_TO_USINT(gu16_Sevcon1_DCLink_VoltageTarget_Tx);
ht_BatteryDemand_Tx.Data[5]	:=	UINT_TO_USINT(SHR(gu16_Sevcon1_DCLink_VoltageTarget_Tx, 8));
ht_BatteryDemand_Tx.Data[6]	:=	gu8_Sevcon1_SEQCurrentLimits;
ht_BatteryDemand_Tx.Data[7]	:=	gu8_Sevcon1_CSCurrentLimits;
ht_BatteryDemand_Tx.Len		:=	8;
	
ht_DirectIControlDemand_Tx.ID		:=	16#191371FA OR EPEC_CANVXD.MASK_29BIT;
ht_DirectIControlDemand_Tx.Data[0]	:=	UINT_TO_USINT(gu16_Sevcon1_DebugIqDirectControl_Tx);
ht_DirectIControlDemand_Tx.Data[1]	:=	UINT_TO_USINT(SHR(gu16_Sevcon1_DebugIqDirectControl_Tx, 8));
ht_DirectIControlDemand_Tx.Data[2]	:=	UINT_TO_USINT(gu16_Sevcon1_DebugIdDirectControl_Tx);
ht_DirectIControlDemand_Tx.Data[3]	:=	UINT_TO_USINT(SHR(gu16_Sevcon1_DebugIdDirectControl_Tx, 8));
ht_DirectIControlDemand_Tx.Data[4]	:=	0;
ht_DirectIControlDemand_Tx.Data[5]	:=	0;
ht_DirectIControlDemand_Tx.Data[6]	:=	gu8_Sevcon1_DirectCurrents;
ht_DirectIControlDemand_Tx.Data[7]	:=	gu8_Sevcon1_CSDirectCurrents;
ht_DirectIControlDemand_Tx.Len		:=	8;
	
hton_SendTimer(IN := TRUE, PT := T#50MS);
IF (hton_SendTimer.Q = TRUE) THEN
	G_CAN2_Channel.SendMessage(i_pMSG:=ADR(ht_TorqueDemand1_Tx));
	G_CAN2_Channel.SendMessage(i_pMSG:=ADR(ht_BatteryDemand_Tx));
	G_CAN2_Channel.SendMessage(i_pMSG:=ADR(ht_DirectIControlDemand_Tx));
	G_CAN2_Channel.SendMessage(i_pMSG:=ADR(ht_TorqueDemand2_Tx));
	hton_SendTimer(IN := FALSE, PT := T#0MS);
END_IF

END_PROGRAM

// Application/UserCode/Sevcon_PSP/Sevcon_Steer_TxConversion
PROGRAM Sevcon_Steer_TxConversion
VAR
END_VAR
VAR CONSTANT
	SEVCON_TX_CF	:	REAL	:=	0.0625;
END_VAR




gu16_Sevcon1_TorqueRq_Tx				:=	REAL_TO_UINT(gr_Sevcon1_TorqueRq / SEVCON_TX_CF);
gu16_Sevcon1_TorqueTractionLimit_Tx		:=	REAL_TO_UINT(gr_Sevcon1_TorqueTractionLimit / SEVCON_TX_CF);
gu16_Sevcon1_TorqueRegenLimit_Tx		:=	REAL_TO_UINT(gr_Sevcon1_TorqueRegenLimit / SEVCON_TX_CF);
gu16_Sevcon1_DCLink_VoltageTarget_Tx	:=	REAL_TO_UINT(gr_Sevcon1_DCLink_VoltageTarget / SEVCON_TX_CF);
gu16_Sevcon1_DebugIqDirectControl_Tx	:=	REAL_TO_UINT(gr_Sevcon1_DebugIqDirectControl / SEVCON_TX_CF);
gu16_Sevcon1_DebugIdDirectControl_Tx	:=	REAL_TO_UINT(gr_Sevcon1_DebugIdDirectControl / SEVCON_TX_CF);

END_PROGRAM

// Application/UserCode/Sevcon_Compressor/Sevcon2_Tx
PROGRAM Sevcon2_Tx
VAR
	ht_TorqueDemand1_Tx			:	EPEC_CANVXD.Msg;
	ht_TorqueDemand2_Tx			:	EPEC_CANVXD.Msg;
	ht_BatteryDemand_Tx			:	EPEC_CANVXD.Msg;
	ht_DirectIControlDemand_Tx	:	EPEC_CANVXD.Msg;
	hton_SendTimer				:	TON;
END_VAR

Sevcon2_TxConversion();

ht_TorqueDemand1_Tx.ID		:=	16#191072FA OR EPEC_CANVXD.MASK_29BIT;
ht_TorqueDemand1_Tx.Data[0]	:=	UINT_TO_USINT(gu16_Sevcon2_TorqueRq_Tx);
ht_TorqueDemand1_Tx.Data[1]	:=	UINT_TO_USINT(SHR(gu16_Sevcon2_TorqueRq_Tx, 8));
ht_TorqueDemand1_Tx.Data[2]	:=	UINT_TO_USINT(gu16_Sevcon2_Controlword);
ht_TorqueDemand1_Tx.Data[3]	:=	UINT_TO_USINT(SHR(gu16_Sevcon2_Controlword, 8));
ht_TorqueDemand1_Tx.Data[4]	:=	UINT_TO_USINT(gu16_Sevcon2_TorqueTractionLimit_Tx);
ht_TorqueDemand1_Tx.Data[5]	:=	UINT_TO_USINT(SHR(gu16_Sevcon2_TorqueTractionLimit_Tx, 8));
ht_TorqueDemand1_Tx.Data[6]	:=	gu8_Sevcon2_SEQCommand1;
ht_TorqueDemand1_Tx.Data[7]	:=	gu8_Sevcon2_CSCommand1;
ht_TorqueDemand1_Tx.Len	:=	8;

ht_TorqueDemand2_Tx.ID		:=	16#191172FA OR EPEC_CANVXD.MASK_29BIT;
ht_TorqueDemand2_Tx.Data[0]	:=	UINT_TO_USINT(gu16_Sevcon2_TorqueRegenLimit_Tx);
ht_TorqueDemand2_Tx.Data[1]	:=	UINT_TO_USINT(SHR(gu16_Sevcon2_TorqueRegenLimit_Tx, 8));
ht_TorqueDemand2_Tx.Data[2]	:=	UINT_TO_USINT(gu16_Sevcon2_SpeedLimitForward);
ht_TorqueDemand2_Tx.Data[3]	:=	UINT_TO_USINT(SHR(gu16_Sevcon2_SpeedLimitForward, 8));
ht_TorqueDemand2_Tx.Data[4]	:=	INT_TO_USINT(gs16_Sevcon2_SpeedLimitReverse);
ht_TorqueDemand2_Tx.Data[5]	:=	INT_TO_USINT(SHR(gs16_Sevcon2_SpeedLimitReverse, 8));
ht_TorqueDemand2_Tx.Data[6]	:=	gu8_Sevcon2_SEQCommand2;
ht_TorqueDemand2_Tx.Data[7]	:=	gu8_Sevcon2_CSCommand2;
ht_TorqueDemand2_Tx.Len		:=	8;

ht_BatteryDemand_Tx.ID		:=	16#191272FA OR EPEC_CANVXD.MASK_29BIT;
ht_BatteryDemand_Tx.Data[0]	:=	UINT_TO_USINT(gu16_Sevcon2_DCLink_ImaxDischarge);
ht_BatteryDemand_Tx.Data[1]	:=	UINT_TO_USINT(SHR(gu16_Sevcon2_DCLink_ImaxDischarge, 8));
ht_BatteryDemand_Tx.Data[2]	:=	INT_TO_USINT(gs16_Sevcon2_DCLink_ImaxRecharge);
ht_BatteryDemand_Tx.Data[3]	:=	INT_TO_USINT(SHR(gs16_Sevcon2_DCLink_ImaxRecharge, 8));
ht_BatteryDemand_Tx.Data[4]	:=	UINT_TO_USINT(gu16_Sevcon2_DCLink_VoltageTarget_Tx);
ht_BatteryDemand_Tx.Data[5]	:=	UINT_TO_USINT(SHR(gu16_Sevcon2_DCLink_VoltageTarget_Tx, 8));
ht_BatteryDemand_Tx.Data[6]	:=	gu8_Sevcon1_SEQCurrentLimits;
ht_BatteryDemand_Tx.Data[7]	:=	gu8_Sevcon1_CSCurrentLimits;
ht_BatteryDemand_Tx.Len		:=	8;
	
ht_DirectIControlDemand_Tx.ID		:=	16#191372FA OR EPEC_CANVXD.MASK_29BIT;
ht_DirectIControlDemand_Tx.Data[0]	:=	UINT_TO_USINT(gu16_Sevcon2_DebugIqDirectControl_Tx);
ht_DirectIControlDemand_Tx.Data[1]	:=	UINT_TO_USINT(SHR(gu16_Sevcon2_DebugIqDirectControl_Tx, 8));
ht_DirectIControlDemand_Tx.Data[2]	:=	UINT_TO_USINT(gu16_Sevcon2_DebugIdDirectControl_Tx);
ht_DirectIControlDemand_Tx.Data[3]	:=	UINT_TO_USINT(SHR(gu16_Sevcon2_DebugIdDirectControl_Tx, 8));
ht_DirectIControlDemand_Tx.Data[4]	:=	0;
ht_DirectIControlDemand_Tx.Data[5]	:=	0;
ht_DirectIControlDemand_Tx.Data[6]	:=	gu8_Sevcon1_DirectCurrents;
ht_DirectIControlDemand_Tx.Data[7]	:=	gu8_Sevcon1_CSDirectCurrents;
ht_DirectIControlDemand_Tx.Len		:=	8;
	
hton_SendTimer(IN := TRUE, PT := T#50MS);
IF (hton_SendTimer.Q = TRUE) THEN
	G_CAN2_Channel.SendMessage(i_pMSG:=ADR(ht_TorqueDemand1_Tx));
	G_CAN2_Channel.SendMessage(i_pMSG:=ADR(ht_BatteryDemand_Tx));
	(*G_CAN2_Channel.SendMessage(i_pMSG:=ADR(ht_DirectIControlDemand_Tx));*)
	G_CAN2_Channel.SendMessage(i_pMSG:=ADR(ht_TorqueDemand2_Tx));
	hton_SendTimer(IN := FALSE, PT := T#0MS);
END_IF

END_PROGRAM

// Application/UserCode/Sevcon_Compressor/Sevcon2_TxConversion
PROGRAM Sevcon2_TxConversion
VAR
END_VAR
VAR CONSTANT
	SEVCON_TX_CF	:	REAL	:=	0.0625;
END_VAR




gu16_Sevcon2_TorqueRq_Tx				:=	REAL_TO_UINT(gr_Sevcon2_TorqueRq / SEVCON_TX_CF);
gu16_Sevcon2_TorqueTractionLimit_Tx		:=	REAL_TO_UINT(gr_Sevcon2_TorqueTractionLimit / SEVCON_TX_CF);
gu16_Sevcon2_TorqueRegenLimit_Tx		:=	REAL_TO_UINT(gr_Sevcon2_TorqueRegenLimit / SEVCON_TX_CF);
gu16_Sevcon2_DCLink_VoltageTarget_Tx	:=	REAL_TO_UINT(gr_Sevcon2_DCLink_VoltageTarget / SEVCON_TX_CF);
gu16_Sevcon2_DebugIqDirectControl_Tx	:=	REAL_TO_UINT(gr_Sevcon2_DebugIqDirectControl / SEVCON_TX_CF);
gu16_Sevcon2_DebugIdDirectControl_Tx	:=	REAL_TO_UINT(gr_Sevcon2_DebugIdDirectControl / SEVCON_TX_CF);

END_PROGRAM

// Application/UserCode/MCU/MCU_Tx
PROGRAM MCU_Tx
VAR
	ht_MCU_VMUComm1_Tx				:	EPEC_CANVXD.Msg;
	ht_MCU_VMUComm2_Tx				:	EPEC_CANVXD.Msg;
	ht_MCU_VMUCommSafety_Tx			:	EPEC_CANVXD.Msg;
	ht_MCU_VMUPollMCU_Tx			:	EPEC_CANVXD.Msg;
	ht_MCU_VMUPollVMUResponse_Tx	:	EPEC_CANVXD.Msg;
	ht_MCU_VMUSelectProtocolVer_Tx	:	EPEC_CANVXD.Msg;
	
	(*Transmit Bytes*)
	hu8_VMUComm1_Byte1				:	USINT;
	hu8_VMUComm1_Byte5				:	USINT;
	hu8_VMUComm1_Byte7				:	USINT;
	
	hu8_VMUComm2_Byte0				:	USINT;
	
	hu8_VMUCommSafety				:	USINT;
	
	hu8_VMUPollMCU_Byte1			:	USINT;
	hu8_VMUPollMCU_Byte2			:	USINT;
	hu8_VMUPollMCU_Byte3			:	USINT;
	hu8_VMUPollMCU_Byte4			:	USINT;
	hu8_VMUPollMCU_Byte5			:	USINT;
	hu8_VMUPollMCU_Byte6			:	USINT;
	hu8_VMUPollMCU_Byte7			:	USINT;
	
	hu8_VMUPollVMUResp_Byte0		:	USINT;
	hu8_VMUPollVMUResp_Byte1		:	USINT;
	hu8_VMUPollVMUResp_Byte2		:	USINT;
	
	(*Transmit Timers*)
	hton_PeriodicSend_Timer			:	TON;
	hton_InitialisationSend_Timer	:	TON;
	
	
END_VAR


MCU_TxConversion();
(*Transmit bytes populating data*)
hu8_VMUComm1_Byte1			:=	(UINT_TO_USINT(SHR(gu16_MCU_MaxChargeCurrent, 8)) AND 2#00001111) +
								(SHL(gu8_MCU_OperationRequest, 5) AND 2#11100000);
hu8_VMUComm1_Byte5			:=	(UINT_TO_USINT(SHR(gu16_MCU_MaxBatteryVoltage, 8)) AND 2#00001111) +
								SHL(BOOL_TO_USINT(gq_MCU_MaxDiscahrgeCurrentStatus), 4) +
								SHL(BOOL_TO_USINT(gq_MCU_MaxBatteryVoltageStatus), 5) +
								SHL(BOOL_TO_USINT(gq_MCU_MinBatteryVoltageStatus), 6) +
								SHL(BOOL_TO_USINT(gq_MCU_MaxChargeCurrentStatus), 7);
hu8_VMUComm1_Byte7			:=	(UINT_TO_USINT(SHR(gu16_MCU_MinBatteryVoltage, 8)) AND 2#00001111) +
								(SHL(gu8_MCU_RollingCounter_VMUComm1, 4) AND 2#11110000);

hu8_VMUComm2_Byte0			:=	(gu8_MCU_OperationalMode_Tx AND 2#00000111) +
								(SHL(gu8_MCU_CommandMode, 3) AND 2#00011000) +
								SHL(BOOL_TO_USINT(gq_MCU_SpeedCommandStatus), 5) +
								SHL(BOOL_TO_USINT(gq_MCU_TorqueCommandStatus), 6);

hu8_VMUCommSafety			:=	(gu8_MCU_ReferenceCommandMode AND 2#00000011) +
								(SHL(gu8_MCU_RollingCounter_VMUCommSafety, 4) AND 2#11110000);

CASE gu8_MCU_VMUPollMCU_Multiplex OF
	MAXMOTORSPEED:								
		hu8_VMUPollMCU_Byte1		:=	UINT_TO_USINT(gu16_MCU_MaxMotorSpeed_Tx);
		hu8_VMUPollMCU_Byte2		:=	UINT_TO_USINT(SHR(gu16_MCU_MaxMotorSpeed_Tx, 8));
		hu8_VMUPollMCU_Byte3		:=	0;
		hu8_VMUPollMCU_Byte4		:=	0;
		hu8_VMUPollMCU_Byte5		:=	0;
		hu8_VMUPollMCU_Byte6		:=	0;
		hu8_VMUPollMCU_Byte7		:=	0;
	MAXMOTORTORQUE:								
		hu8_VMUPollMCU_Byte1		:=	UINT_TO_USINT(gu16_MCU_MaxMotorTorque_Tx);
		hu8_VMUPollMCU_Byte2		:=	UINT_TO_USINT(SHR(gu16_MCU_MaxMotorTorque_Tx, 8));
		hu8_VMUPollMCU_Byte3		:=	0;
		hu8_VMUPollMCU_Byte4		:=	0;
		hu8_VMUPollMCU_Byte5		:=	0;
		hu8_VMUPollMCU_Byte6		:=	0;
		hu8_VMUPollMCU_Byte7		:=	0;
	PROTOCOLVERSION:								
		hu8_VMUPollMCU_Byte1		:=	gu8_MCU_MajorMCUProtocol_Tx;
		hu8_VMUPollMCU_Byte2		:=	gu8_MCU_MinorMCUProtocol_Tx;
		hu8_VMUPollMCU_Byte3		:=	0;
		hu8_VMUPollMCU_Byte4		:=	0;
		hu8_VMUPollMCU_Byte5		:=	0;
		hu8_VMUPollMCU_Byte6		:=	0;
		hu8_VMUPollMCU_Byte7		:=	0;
	SWVERSION1:								
		hu8_VMUPollMCU_Byte1		:=	gu8_MCU_MajorMCUSW_Tx;
		hu8_VMUPollMCU_Byte2		:=	gu8_MCU_MinorMCUSW_Tx;
		hu8_VMUPollMCU_Byte3		:=	UINT_TO_USINT(gu16_MCU_BranchMCUSW_Tx);
		hu8_VMUPollMCU_Byte4		:=	UINT_TO_USINT(SHR(gu16_MCU_BranchMCUSW_Tx, 8));
		hu8_VMUPollMCU_Byte5		:=	0;
		hu8_VMUPollMCU_Byte6		:=	0;
		hu8_VMUPollMCU_Byte7		:=	0;
	SWVERSION2:								
		hu8_VMUPollMCU_Byte1		:=	UDINT_TO_USINT(gu32_MCU_RevisionMCUSW_Tx);
		hu8_VMUPollMCU_Byte2		:=	UDINT_TO_USINT(SHR(gu32_MCU_RevisionMCUSW_Tx, 8));
		hu8_VMUPollMCU_Byte3		:=	UDINT_TO_USINT(SHR(gu32_MCU_RevisionMCUSW_Tx, 16));
		hu8_VMUPollMCU_Byte4		:=	UDINT_TO_USINT(SHR(gu32_MCU_RevisionMCUSW_Tx, 24));
		hu8_VMUPollMCU_Byte5		:=	0;
		hu8_VMUPollMCU_Byte6		:=	0;
		hu8_VMUPollMCU_Byte7		:=	0;
	TOTALMOTORROTATION:								
		hu8_VMUPollMCU_Byte1		:=	(*UDINT_TO_USINT(gu32_MCU_TotalMotorRotation_LSB_Tx)*)0;
		hu8_VMUPollMCU_Byte2		:=	(*UDINT_TO_USINT(SHR(gu32_MCU_TotalMotorRotation_LSB_Tx, 8))*)0;
		hu8_VMUPollMCU_Byte3		:=	(*UDINT_TO_USINT(SHR(gu32_MCU_TotalMotorRotation_LSB_Tx, 16))*)0;
		hu8_VMUPollMCU_Byte4		:=	(*UDINT_TO_USINT(SHR(gu32_MCU_TotalMotorRotation_LSB_Tx, 24))*)0;
		hu8_VMUPollMCU_Byte5		:=	(*UDINT_TO_USINT(gu32_MCU_TotalMotorRotation_MSB_Tx)*)0;
		hu8_VMUPollMCU_Byte6		:=	(*UDINT_TO_USINT(SHR(gu32_MCU_TotalMotorRotation_MSB_Tx, 8))*)0;
		hu8_VMUPollMCU_Byte7		:=	0;
	TOTALMOTORROTATIONUSINTMCU:								
		hu8_VMUPollMCU_Byte1		:=	0;
		hu8_VMUPollMCU_Byte2		:=	0;
		hu8_VMUPollMCU_Byte3		:=	0;
		hu8_VMUPollMCU_Byte4		:=	0;
		hu8_VMUPollMCU_Byte5		:=	0;
		hu8_VMUPollMCU_Byte6		:=	0;
		hu8_VMUPollMCU_Byte7		:=	0;
END_CASE

hu8_VMUPollVMUResp_Byte0	:=		(gu8_MCU_PollVMUResponse_Multiplex AND 2#01111111) +
									SHL(BOOL_TO_USINT(gq_MCU_PollVMUResponse_Acknowledgement), 7);
CASE gu8_MCU_PollVMUResponse_Multiplex OF
	VMUBOOTNUMBER:
		hu8_VMUPollVMUResp_Byte1	:=	UINT_TO_USINT(gu16_MCU_BootNumber);
		hu8_VMUPollVMUResp_Byte2	:=	UINT_TO_USINT(SHR(gu16_MCU_BootNumber, 8));
END_CASE
								
								
ht_MCU_VMUComm1_Tx.ID		:=	16#040;
ht_MCU_VMUComm1_Tx.Data[0]	:=	UINT_TO_USINT(gu16_MCU_MaxChargeCurrent);
ht_MCU_VMUComm1_Tx.Data[1]	:=	hu8_VMUComm1_Byte1;
ht_MCU_VMUComm1_Tx.Data[2]	:=	UINT_TO_USINT(gu16_MCU_MaxDischargeCurrent);
ht_MCU_VMUComm1_Tx.Data[3]	:=	UINT_TO_USINT(SHR(gu16_MCU_MaxDischargeCurrent, 8)) AND 2#00001111;
ht_MCU_VMUComm1_Tx.Data[4]	:=	UINT_TO_USINT(gu16_MCU_MaxBatteryVoltage);
ht_MCU_VMUComm1_Tx.Data[5]	:=	hu8_VMUComm1_Byte5;
ht_MCU_VMUComm1_Tx.Data[6]	:=	UINT_TO_USINT(gu16_MCU_MinBatteryVoltage);
ht_MCU_VMUComm1_Tx.Data[7]	:=	hu8_VMUComm1_Byte7;
ht_MCU_VMUComm1_Tx.Len		:=	8;

ht_MCU_VMUComm2_Tx.ID		:=	16#041;
ht_MCU_VMUComm2_Tx.Data[0]	:=	hu8_VMUComm2_Byte0;
ht_MCU_VMUComm2_Tx.Data[1]	:=	UINT_TO_USINT(gu16_MCU_TorqueCommand_Tx);
ht_MCU_VMUComm2_Tx.Data[2]	:=	UINT_TO_USINT(SHR(gu16_MCU_TorqueCommand_Tx, 8));
ht_MCU_VMUComm2_Tx.Data[3]	:=	UINT_TO_USINT(gu16_MCU_SpeedCommand_Tx);
ht_MCU_VMUComm2_Tx.Data[4]	:=	UINT_TO_USINT(SHR(gu16_MCU_SpeedCommand_Tx, 8));
ht_MCU_VMUComm2_Tx.Data[5]	:=	SHL(gu8_MCU_RollingCounter_VMUComm2, 4);
ht_MCU_VMUComm2_Tx.Data[6]	:=	0;
ht_MCU_VMUComm2_Tx.Data[7]	:=	0;
ht_MCU_VMUComm2_Tx.Len		:=	6;

ht_MCU_VMUCommSafety_Tx.ID		:=	16#042;
ht_MCU_VMUCommSafety_Tx.Data[0]	:=	UINT_TO_USINT(gu16_MCU_ReferenceTorqueCommand_Tx);
ht_MCU_VMUCommSafety_Tx.Data[1]	:=	UINT_TO_USINT(SHR(gu16_MCU_ReferenceTorqueCommand_Tx, 8));
ht_MCU_VMUCommSafety_Tx.Data[2]	:=	UINT_TO_USINT(gu16_MCU_ReferenceSpeedCommand_Tx);
ht_MCU_VMUCommSafety_Tx.Data[3]	:=	UINT_TO_USINT(SHR(gu16_MCU_ReferenceSpeedCommand_Tx, 8));
ht_MCU_VMUCommSafety_Tx.Data[4]	:=	hu8_VMUCommSafety;
ht_MCU_VMUCommSafety_Tx.Data[5]	:=	0;
ht_MCU_VMUCommSafety_Tx.Data[6]	:=	0;
ht_MCU_VMUCommSafety_Tx.Data[7]	:=	0;
ht_MCU_VMUCommSafety_Tx.Len		:=	5;

ht_MCU_VMUPollMCU_Tx.ID		:=	16#447;
ht_MCU_VMUPollMCU_Tx.Data[0]	:=	gu8_MCU_VMUPollMCU_Multiplex AND 2#01111111;
ht_MCU_VMUPollMCU_Tx.Data[1]	:=	hu8_VMUPollMCU_Byte1;
ht_MCU_VMUPollMCU_Tx.Data[2]	:=	hu8_VMUPollMCU_Byte2;
ht_MCU_VMUPollMCU_Tx.Data[3]	:=	hu8_VMUPollMCU_Byte3;
ht_MCU_VMUPollMCU_Tx.Data[4]	:=	hu8_VMUPollMCU_Byte4;
ht_MCU_VMUPollMCU_Tx.Data[5]	:=	hu8_VMUPollMCU_Byte5;
ht_MCU_VMUPollMCU_Tx.Data[6]	:=	hu8_VMUPollMCU_Byte6;
ht_MCU_VMUPollMCU_Tx.Data[7]	:=	hu8_VMUPollMCU_Byte7;
ht_MCU_VMUPollMCU_Tx.Len		:=	8;

ht_MCU_VMUPollVMUResponse_Tx.ID		:=	16#446;
ht_MCU_VMUPollVMUResponse_Tx.Data[0]	:=	hu8_VMUPollVMUResp_Byte0;
ht_MCU_VMUPollVMUResponse_Tx.Data[1]	:=	hu8_VMUPollVMUResp_Byte1;
ht_MCU_VMUPollVMUResponse_Tx.Data[2]	:=	hu8_VMUPollVMUResp_Byte2;
ht_MCU_VMUPollVMUResponse_Tx.Data[3]	:=	0;
ht_MCU_VMUPollVMUResponse_Tx.Data[4]	:=	0;
ht_MCU_VMUPollVMUResponse_Tx.Data[5]	:=	0;
ht_MCU_VMUPollVMUResponse_Tx.Data[6]	:=	0;
ht_MCU_VMUPollVMUResponse_Tx.Data[7]	:=	0;
ht_MCU_VMUPollVMUResponse_Tx.Len		:=	8;

ht_MCU_VMUSelectProtocolVer_Tx.ID		:=	16#444;
ht_MCU_VMUSelectProtocolVer_Tx.Data[0]	:=	gu8_MCU_SelectMajorMCUProtocol_Tx;
ht_MCU_VMUSelectProtocolVer_Tx.Data[1]	:=	gu8_MCU_SelectMinorMCUProtocol_Tx;
ht_MCU_VMUSelectProtocolVer_Tx.Data[2]	:=	0;
ht_MCU_VMUSelectProtocolVer_Tx.Data[3]	:=	0;
ht_MCU_VMUSelectProtocolVer_Tx.Data[4]	:=	0;
ht_MCU_VMUSelectProtocolVer_Tx.Data[5]	:=	0;
ht_MCU_VMUSelectProtocolVer_Tx.Data[6]	:=	0;
ht_MCU_VMUSelectProtocolVer_Tx.Data[7]	:=	0;
ht_MCU_VMUSelectProtocolVer_Tx.Len		:=	2;


IF (gu8_MCU_MajorMCUProtocol = 0(* AND gq_InitialProtocolGrab = FALSE*)) THEN
	hton_InitialisationSend_Timer(IN := NOT(hton_InitialisationSend_Timer.Q), PT := T#10MS);
	IF (hton_InitialisationSend_Timer.Q = TRUE) THEN
		G_CAN1_Channel.SendMessage(i_pMSG:=ADR(ht_MCU_VMUSelectProtocolVer_Tx));
	END_IF
ELSIF (gu8_MCU_MajorMCUProtocol <> 0) THEN
	(*hton_PeriodicSend_Timer(IN := TRUE, PT := T#10MS);*)
	IF (hton_PeriodicSend_Timer.Q = (*TRUE*)FALSE) THEN
		G_CAN1_Channel.SendMessage(i_pMSG:=ADR(ht_MCU_VMUComm1_Tx));
		G_CAN1_Channel.SendMessage(i_pMSG:=ADR(ht_MCU_VMUComm2_Tx));
		G_CAN1_Channel.SendMessage(i_pMSG:=ADR(ht_MCU_VMUCommSafety_Tx));
		IF (gu8_MCU_VMUPollMCU_Multiplex >= 0 AND gu8_MCU_VMUPollMCU_Multiplex < 8) THEN
			G_CAN1_Channel.SendMessage(i_pMSG:=ADR(ht_MCU_VMUPollMCU_Tx));
		END_IF
		gu8_MCU_RollingCounter_VMUComm1			:=	gu8_MCU_RollingCounter_VMUComm1 + 1;
		gu8_MCU_RollingCounter_VMUComm2			:=	gu8_MCU_RollingCounter_VMUComm2 + 1;
		gu8_MCU_RollingCounter_VMUCommSafety	:=	gu8_MCU_RollingCounter_VMUCommSafety + 1;
		IF (gu8_MCU_RollingCounter_VMUComm1 > 15) THEN
			gu8_MCU_RollingCounter_VMUComm1	:=	0;
		END_IF
		IF (gu8_MCU_RollingCounter_VMUComm2 > 15) THEN
			gu8_MCU_RollingCounter_VMUComm2	:=	0;
		END_IF
		IF (gu8_MCU_RollingCounter_VMUCommSafety > 15) THEN
			gu8_MCU_RollingCounter_VMUCommSafety	:=	0;
		END_IF
		(*Update the last command value sent*)
		gr_MCU_PreviousTorqueCommand		:=	gr_MCU_TorqueCommand_Limited;
		hton_PeriodicSend_Timer(IN := FALSE, PT := T#0MS);
	END_IF
	gq_InitialProtocolGrab	:=	TRUE;
END_IF

END_PROGRAM

// Application/UserCode/MCU/MCU_TxConversion
PROGRAM MCU_TxConversion
VAR
	hr_MCU_LowerLimitTorqueCommand	:	REAL;
	hr_MCU_UpperLimitTorqueCommand	:	REAL;
	LowPassFilter	:	OSCAT_BASIC.FT_PT1;
	TimeConstant	:	REAL	:=	1000;
END_VAR
VAR RETAIN
	hr_INCREASETORQUERAMP	:	REAL	:=	3500; (*Nm/s*)
	hr_DECREASETORQUERAMP	:	REAL	:=	7000; (*Nm/s*)
END_VAR


(*10ms *)
(*
hr_MCU_LowerLimitTorqueCommand		:=	gr_MCU_PreviousTorqueCommand - (hr_DECREASETORQUERAMP / 100);
hr_MCU_UpperLimitTorqueCommand		:=	gr_MCU_PreviousTorqueCommand + (hr_INCREASETORQUERAMP / 100);
gr_MCU_TorqueCommand_Limited		:=	LIMIT(hr_MCU_LowerLimitTorqueCommand, gr_MCU_TorqueCommand_PreCF_Limited, hr_MCU_UpperLimitTorqueCommand);
*)
LowPassFilter(in := gr_MCU_TorqueCommand_PreCF_Limited, T := REAL_TO_TIME(TimeConstant), K := 1, out => gr_MCU_TorqueCommand_Limited);


gu16_MCU_TorqueCommand_Tx			:=	REAL_TO_UINT((gr_MCU_TorqueCommand_Limited + 4096) / 0.125);
gu16_MCU_SpeedCommand_Tx			:=	REAL_TO_UINT(gr_MCU_SpeedCommand_PreCF) + 32767;
gu16_MCU_ReferenceTorqueCommand_Tx	:=	REAL_TO_UINT((gr_MCU_ReferenceTorqueCommand_PreCF + 4096) / 0.125);
gu16_MCU_ReferenceSpeedCommand_Tx	:=	REAL_TO_UINT(gr_MCU_ReferenceSpeedCommand_PreCF) + 32767;
gu16_MCU_MaxMotorSpeed_Tx			:=	REAL_TO_UINT(gr_MCU_MaxMotorSpeed_PreCF + 32767);
gu16_MCU_MaxMotorTorque_Tx			:=	REAL_TO_UINT(4000 / 0.125); (*Not currently sent as the max torque is gained from the MCU*)

gu8_MCU_SelectMajorMCUProtocol_Tx	:=	4;
gu8_MCU_SelectMinorMCUProtocol_Tx	:=	0;

END_PROGRAM

// Application/UserCode/CAN4/CAN4_Tx
PROGRAM CAN4_Tx
VAR
	ht_CAN4_601_Tx	:	EPEC_CANVXD.Msg;
	ht_CAN4_201_Tx	:	EPEC_CANVXD.Msg;
	ht_CAN4_301_Tx	:	EPEC_CANVXD.Msg;
	ht_CAN4_401_Tx	:	EPEC_CANVXD.Msg;
	ht_CAN4_8DD1_Tx	: 	EPEC_CANVXD.Msg;
	hton_MessageSend_Timer	:	TON;
	ht_ETC2_Tx	:	EPEC_CANVXD.Msg;
	NMT1_Tx	:	EPEC_CANVXD.Msg;
	Dash_FF02_Tx : EPEC_CANVXD.Msg;
	Dash_FF04_Tx : EPEC_CANVXD.Msg;
	Dash_FF08_Tx	:	EPEC_CANVXD.Msg;
	Dash_FF12_Tx	:	EPEC_CANVXD.Msg;
	Dash_FF14_Tx	:	EPEC_CANVXD.Msg;
	Dash_FF21_Tx	:	EPEC_CANVXD.Msg;
	Tx_Timer	:	TON;
	hu8_Temp	:	USINT := 10;
	
	Version: STRING;
	
END_VAR

CAN4_TxConversion();
BMS_to_HMI();
DCDC_to_HMI();
MCU_to_HMI();
Sevcon_to_HMI();
VMU_to_HMI();
IF gq_CAN4_ChargerPP_Tx THEN BRUSA_to_HMI();
END_IF
Version := Project_Infomation.ver;
 
//* special needs for HMI
ht_CAN4_8DD1_Tx.ID		:=	16#188000DD OR EPEC_CANVXD.MASK_29BIT;
ht_CAN4_8DD1_Tx.Data[0]	:=	gu8_ChassisType;
ht_CAN4_8DD1_Tx.Data[1].0	:=	gq_Frosty_NoWheelSpeedSensors;
ht_CAN4_8DD1_Tx.Data[1].1	:=	gq_BodyStepInstalled;
ht_CAN4_8DD1_Tx.Data[1].2	:=	gq_Daimler_PowerShift_Installed;
ht_CAN4_8DD1_Tx.Data[1].3	:=	gq_APU_Installed;
ht_CAN4_8DD1_Tx.Data[1].4	:=	0;//gq_RearSteer_Installed; Not Used Spare
ht_CAN4_8DD1_Tx.Data[1].5	:=	gq_CAN1_Merc_Gears;
ht_CAN4_8DD1_Tx.Data[1].6	:=	E_Stop_Installed;
ht_CAN4_8DD1_Tx.Data[1].7	:=	DO_q_HeaterOut_DI;
ht_CAN4_8DD1_Tx.Data[2] :=	Project_Infomation.Major;
ht_CAN4_8DD1_Tx.Data[3]	:=	Project_Infomation.Minor;
ht_CAN4_8DD1_Tx.Data[4]	:=	Project_Infomation.patch;
ht_CAN4_8DD1_Tx.Data[5]	:=	0;
ht_CAN4_8DD1_Tx.Data[6]	:=	0;
ht_CAN4_8DD1_Tx.Data[7]	:=	0;
ht_CAN4_8DD1_Tx.Len		:=	8;

(***************************************************************************)
ht_CAN4_601_Tx.ID		:=	16#601;
ht_CAN4_601_Tx.Data[0]	:=	UINT_TO_USINT(gu16_CAN4_TripCounter_km_Tx);
ht_CAN4_601_Tx.Data[1]	:=	UINT_TO_USINT(SHR(gu16_CAN4_TripCounter_km_Tx, 8));
ht_CAN4_601_Tx.Data[2]	:=	SINT_TO_USINT(gs8_CAN4_CruiseControlSetpoint_Tx);
ht_CAN4_601_Tx.Data[3]	:=	INT_TO_USINT(gs16_CAN4_PowerIndication_Tx);
ht_CAN4_601_Tx.Data[4]	:=	INT_TO_USINT(SHR(gs16_CAN4_PowerIndication_Tx, 8));
ht_CAN4_601_Tx.Data[5]	:=	SINT_TO_USINT(gs8_CAN4_DummyScreen601_Tx);		
ht_CAN4_601_Tx.Data[6]	:=	0;		
ht_CAN4_601_Tx.Data[7]	:=	0;		
ht_CAN4_601_Tx.Len		:=	8;

ht_CAN4_201_Tx.ID		:=	16#201;
ht_CAN4_201_Tx.Data[0]	:=	SINT_TO_USINT(gs8_CAN4_DisplayTemp_Tx);
ht_CAN4_201_Tx.Data[1]	:=	SINT_TO_USINT(gs8_CAN4_DisplayDirection_Tx);
ht_CAN4_201_Tx.Data[2]	:=	SINT_TO_USINT(gs8_CAN4_SOC_Tx);
ht_CAN4_201_Tx.Data[3]	:=	SINT_TO_USINT(gs8_CAN4_DispVehicleStatus_Tx);
ht_CAN4_201_Tx.Data[4]	:=	SINT_TO_USINT(gs8_CAN4_PowerIndicationRelative_Tx);
ht_CAN4_201_Tx.Data[5]	:=	SINT_TO_USINT(gs8_CAN4_DisplayStatus_Tx);
ht_CAN4_201_Tx.Data[6]	:=	SINT_TO_USINT(gs8_CAN4_SOC1_Tx);
ht_CAN4_201_Tx.Data[7]	:=	SINT_TO_USINT(gs8_CAN4_BatteryVoltage_Tx);
ht_CAN4_201_Tx.Len		:=	8;

ht_CAN4_301_Tx.ID		:=	16#301;
ht_CAN4_301_Tx.Data[0]	:=	INT_TO_USINT(gs16_CAN4_BatteryCurrent_Tx);
ht_CAN4_301_Tx.Data[1]	:=	INT_TO_USINT(SHR(gs16_CAN4_BatteryCurrent_Tx, 8));
ht_CAN4_301_Tx.Data[2]	:=	UINT_TO_USINT(gu16_CAN4_DisplayRangeMin_Tx);
ht_CAN4_301_Tx.Data[3]	:=	UINT_TO_USINT(SHR(gu16_CAN4_DisplayRangeMin_Tx, 8));
ht_CAN4_301_Tx.Data[4]	:=	UINT_TO_USINT(gu16_BMS1_LowCellVoltage); (*gu8_BMS1_LowCellV_Tx*)
ht_CAN4_301_Tx.Data[5]	:=	UINT_TO_USINT(SHR(gu16_BMS1_LowCellVoltage, 8)); (*gu8_BMS2_LowCellV_Tx*)
ht_CAN4_301_Tx.Data[6]	:=	UINT_TO_USINT(gu16_BMS2_LowCellVoltage);
ht_CAN4_301_Tx.Data[7]	:=	UINT_TO_USINT(SHR(gu16_BMS2_LowCellVoltage, 8));
ht_CAN4_301_Tx.Len		:=	8;

ht_CAN4_401_Tx.ID		:=	16#401;
ht_CAN4_401_Tx.Data[0]	:=	SINT_TO_USINT(gs8_CAN4_MotorTemp_Tx);
ht_CAN4_401_Tx.Data[1]	:=	SINT_TO_USINT(gs8_CAN4_InverterTemp_Tx);
ht_CAN4_401_Tx.Data[2]	:=	gu8_CAN4_ChargerStatus_Tx;
ht_CAN4_401_Tx.Data[3]	:=	SINT_TO_USINT(gs8_CAN4_ThrottlePedal_Tx);
ht_CAN4_401_Tx.Data[4]	:=	gu8_Compressor_Temp_To_Screen;
ht_CAN4_401_Tx.Data[5]	:=	SINT_TO_USINT(gs8_CAN4_VehicleSpeedMsg_Tx);
ht_CAN4_401_Tx.Data[6]	:=	SINT_TO_USINT(gs8_CAN4_VehicleStatus_Tx);
ht_CAN4_401_Tx.Data[7]	:=	SINT_TO_USINT(gs8_CAN4_RegenTorquePercDisplay_Tx);
ht_CAN4_401_Tx.Len		:=	8;
(***************************************************************************)


ht_ETC2_Tx.ID		:=	16#18F00503 OR EPEC_CANVXD.MASK_29BIT;
ht_ETC2_Tx.Data[0]	:=	gu8_CurrentGear2; (*Current Gear2*)
ht_ETC2_Tx.Data[1]	:=	UINT_TO_USINT(gu16_CurrentGear); (*Current Gear LSB*)
ht_ETC2_Tx.Data[2]	:=	UINT_TO_USINT(SHR(gu16_CurrentGear, 8)); (*Current Gear MSB*)
ht_ETC2_Tx.Data[3]	:=	gu8_CurrentGear2; (*Current Gear2*)
ht_ETC2_Tx.Data[4]	:=	16#FF;
ht_ETC2_Tx.Data[5]	:=	16#FF;
ht_ETC2_Tx.Data[6]	:=	UINT_TO_USINT(gu16_CurrentGear1); (*Current Gear1 LSB*)
ht_ETC2_Tx.Data[7]	:=	UINT_TO_USINT(SHR(gu16_CurrentGear1, 8)); (*Current Gear1 MSB*)
ht_ETC2_Tx.Len		:=	8;

NMT1_Tx.ID		:=	0;
NMT1_Tx.Data[0]	:=	1;
NMT1_Tx.Data[1]	:=	0;
NMT1_Tx.Len		:=	2;

Dash_FF08_Tx.ID	:=	16#18FF08C4 OR EPEC_CANVXD.MASK_29BIT;
Dash_FF08_Tx.Data[0].0	:=	DO_q_DrivetrainCoolingFan_DO;
Dash_FF08_Tx.Data[0].1	:=	gq_Dash_Sevcon1_Enable;
Dash_FF08_Tx.Data[0].2	:=	gq_Dash_Sevcon2_Enable;
Dash_FF08_Tx.Data[0].3	:=	DO_q_DrivetrainDCDCInhibit_DO;
Dash_FF08_Tx.Data[0].4	:=	Brusa1_Rx.S_ProximityDet;
Dash_FF08_Tx.Data[0].5	:=	DO_q_Battery1ChargePrecharge_DO;
Dash_FF08_Tx.Data[0].6	:=	DO_q_Battery1ChargeMain_DO;
Dash_FF08_Tx.Data[0].7	:=	DO_q_Battery2ChargePrecharge_DO;
Dash_FF08_Tx.Data[1].0	:=	DO_q_Battery2ChargeMain_DO;
Dash_FF08_Tx.Data[1].1	:=	gq_Dash_Charge_Rq;
Dash_FF08_Tx.Data[1].2	:=	gq_Dash_Discharge_Rq;
Dash_FF08_Tx.Data[1].3	:=	gq_Dash_Charge_Rq;
Dash_FF08_Tx.Data[1].4	:=	gq_Dash_Discharge_Rq;
Dash_FF08_Tx.Data[1].5	:=	DI_q_VehicleKL15_DI;
Dash_FF08_Tx.Data[1].6	:=	DO_q_ChargePlugLED_Red_DO;
Dash_FF08_Tx.Data[1].7	:=	DO_q_ChargePlugLED_Green_DO;
Dash_FF08_Tx.Data[2]	:=	gu8_SystemState; (*Might need to change this*)
Dash_FF08_Tx.Data[3]	:=	REAL_TO_USINT(gr_VehicleSpeed_kmph);
Dash_FF08_Tx.Data[4]	:=	gu8_BMS_SOC;
Dash_FF08_Tx.Data[5]	:=	INT_TO_USINT(gs16_Dash_BattCurrent_Tx);
Dash_FF08_Tx.Data[6]	:=	INT_TO_USINT(SHR(gs16_Dash_BattCurrent_Tx, 8));
Dash_FF08_Tx.Data[7].0	:=	DO_q_BatteryDischargePrecharge_DO;
Dash_FF08_Tx.Data[7].1	:=	DO_q_BatteryDischargeMain_DO;
Dash_FF08_Tx.Len	:=	8;

Dash_FF12_Tx.ID	:=	16#18FF12C4 OR EPEC_CANVXD.MASK_29BIT;
Dash_FF12_Tx.Data[0].0	:=	DI_q_VehicleKL15_DI;
Dash_FF12_Tx.Data[0].1	:=	FALSE; (*Crawl*)
Dash_FF12_Tx.Data[0].2	:=	gq_BrakeSwitch;
Dash_FF12_Tx.Data[0].3	:=	gq_HandBrake;
Dash_FF12_Tx.Data[0].4	:=	gq_BattFullyCharged;
Dash_FF12_Tx.Data[0].5	:=	gq_Heater_EnableBit;
Dash_FF12_Tx.Data[0].6	:=	FALSE; (*DI AC*)
Dash_FF12_Tx.Data[0].7	:=	DO_q_ChargePlugLED_Blue_DO;
Dash_FF12_Tx.Data[1]	:=	gu8_CurrentGear2;
Dash_FF12_Tx.Data[2]	:=	gu8_Dash_AccelPedal_Tx;
Dash_FF12_Tx.Data[3]	:=	hu8_Temp; (*Inverter Temp*)
Dash_FF12_Tx.Data[4]	:=	gu8_Dash_BrakePressure1_Tx;
Dash_FF12_Tx.Data[5]	:=	gu8_Dash_BrakePressure2_Tx;
Dash_FF12_Tx.Data[6]	:=	INT_TO_USINT(gs16_Dash_Power);
Dash_FF12_Tx.Data[7]	:=	INT_TO_USINT(SHR(gs16_Dash_Power, 8));
Dash_FF12_Tx.Len	:=	8;
(*
(*BMS*)
Dash_FF02_Tx.ID	:=	16#18FF02C4;
Dash_FF02_Tx.Data[0]	:=	REAL_TO_USINT(gr_BMS_BatteryVoltage);
Dash_FF02_Tx.Data[1]	:=	UINT_TO_USINT(SHR(REAL_TO_UINT(gr_BMS_BatteryVoltage), 8));
Dash_FF02_Tx.Data[2]	:=	UINT_TO_USINT(gu16_BMS1_LowCellVoltage);
Dash_FF02_Tx.Data[3]	:=	UINT_TO_USINT(SHR(gu16_BMS1_LowCellVoltage, 8));
Dash_FF02_Tx.Data[4]	:=	UINT_TO_USINT(gu16_BMS1_HighCellVoltage);
Dash_FF02_Tx.Data[5]	:=	UINT_TO_USINT(SHR(gu16_BMS1_HighCellVoltage, 8));
Dash_FF02_Tx.Data[6]	:=	UINT_TO_USINT(gu16_BMS1_LowCellVoltage_ID);
Dash_FF02_Tx.Data[7]	:=	UINT_TO_USINT(gu16_BMS1_HighCellVoltage_ID);
Dash_FF02_Tx.Len	:=	8;
Dash_FF04_Tx.ID	:=	16#18FF04C4;
Dash_FF04_Tx.Data[0]	:=	REAL_TO_USINT(gr_BMS_DCL);
Dash_FF04_Tx.Data[1]	:=	UINT_TO_USINT(SHR(REAL_TO_UINT(gr_BMS_DCL), 8));
Dash_FF04_Tx.Data[2]	:=	INT_TO_USINT(gs16_BMS_BatteryCurrent);
Dash_FF04_Tx.Data[3]	:=	INT_TO_USINT(SHR(REAL_TO_INT(gs16_BMS_BatteryCurrent), 8));
Dash_FF04_Tx.Data[4]	:=	REAL_TO_USINT(gr_BMS1_Voltage);
Dash_FF04_Tx.Data[5]	:=	UINT_TO_USINT(SHR(REAL_TO_UINT(gr_BMS1_Voltage), 8));
Dash_FF04_Tx.Data[6]	:=	REAL_TO_USINT(gr_BMS_CCL);
Dash_FF04_Tx.Data[7]	:=	UINT_TO_USINT(SHR(REAL_TO_UINT(gr_BMS_CCL), 8));
Dash_FF04_Tx.Len	:=	8;
Dash_FF21_Tx.ID	:=	16#18FF21C4;
Dash_FF21_Tx.Data[0]	:=	gu8_BMS_LowTemp_ID;
Dash_FF21_Tx.Data[1]	:=	gu8_BMS_HighTemp_ID;
Dash_FF21_Tx.Data[2]	:=	SINT_TO_USINT(gs8_Dash_AverageTemp_Tx);
Dash_FF21_Tx.Data[3]	:=	SINT_TO_USINT(gs8_Dash_HighTemp_Tx);
Dash_FF21_Tx.Data[4]	:=	SINT_TO_USINT(gs8_Dash_LowTemp_Tx);
Dash_FF21_Tx.Data[5]	:=	gu8_BMS_SOC;
Dash_FF21_Tx.Data[6]	:=	0;
Dash_FF21_Tx.Data[7]	:=	0;
Dash_FF21_Tx.Len	:=	8;	
*)

Dash_FF14_Tx.ID	:=	16#18FF14C4 OR EPEC_CANVXD.MASK_29BIT;
Dash_FF14_Tx.Data[0]	:=	INT_TO_USINT(gs16_Sevcon1_SpeedMeasured);
Dash_FF14_Tx.Data[1]	:=	INT_TO_USINT(SHR(gs16_Sevcon1_SpeedMeasured, 8));
Dash_FF14_Tx.Data[2]	:=	INT_TO_USINT(gs16_Sevcon2_SpeedMeasured);
Dash_FF14_Tx.Data[3]	:=	INT_TO_USINT(SHR(gs16_Sevcon2_SpeedMeasured, 8));
Dash_FF14_Tx.Data[5]	:=	REAL_TO_USINT(gr_Sevcon1_DCLink_Voltage);
Dash_FF14_Tx.Data[4]	:=	UINT_TO_USINT(SHR(REAL_TO_UINT(gr_Sevcon1_DCLink_Voltage * 16), 8));
Dash_FF14_Tx.Data[7]	:=	REAL_TO_USINT(gr_Sevcon2_DCLink_Voltage);
Dash_FF14_Tx.Data[6]	:=	UINT_TO_USINT(SHR(REAL_TO_UINT(gr_Sevcon2_DCLink_Voltage  *16), 8));
Dash_FF14_Tx.Len	:=	8;

(*FA00 new address to start on, choose an appropriate source address for the controller*)


hton_MessageSend_Timer(IN := NOT(hton_MessageSend_Timer.Q), PT := T#100MS);
IF (hton_MessageSend_Timer.Q = TRUE) THEN
	G_CAN4_Channel.SendMessage(i_pMSG:=ADR(ht_ETC2_Tx));
	(*Dash Screen*)
	G_CAN4_Channel.SendMessage(i_pMSG:=ADR(Dash_FF08_Tx));
	G_CAN4_Channel.SendMessage(i_pMSG:=ADR(Dash_FF12_Tx));
	G_CAN4_Channel.SendMessage(i_pMSG:=ADR(Dash_FF14_Tx));
	
	(*G_CAN4_Channel.SendMessage(i_pMSG:=ADR(Dash_FF08_Tx));
	G_CAN4_Channel.SendMessage(i_pMSG:=ADR(Dash_FF04_Tx));
	G_CAN4_Channel.SendMessage(i_pMSG:=ADR(Dash_FF02_Tx));
	G_CAN4_Channel.SendMessage(i_pMSG:=ADR(Dash_FF21_Tx));*)

END_IF
Tx_Timer(IN := NOT(Tx_Timer.Q), PT := T#1000MS);
IF (Tx_Timer.Q = TRUE) THEN
	G_CAN4_Channel.SendMessage(i_pMSG:=ADR(NMT1_Tx));
	
	G_CAN4_Channel.SendMessage(i_pMSG:=ADR(ht_CAN4_601_Tx));
	G_CAN4_Channel.SendMessage(i_pMSG:=ADR(ht_CAN4_201_Tx));
	G_CAN4_Channel.SendMessage(i_pMSG:=ADR(ht_CAN4_301_Tx));
	G_CAN4_Channel.SendMessage(i_pMSG:=ADR(ht_CAN4_401_Tx));
	G_CAN4_Channel.SendMessage(i_pMSG:=ADR(ht_CAN4_8DD1_Tx));
	
END_IF

END_PROGRAM

// Application/UserCode/CAN4/CAN4_TxConversion
PROGRAM CAN4_TxConversion
VAR
	(*Vehicle Direction (FORWARD := 16#7E, NEUTRAL := 16#7D, REVERSE := 16#7C, UNKNOWN := 16#00)*)
END_VAR
VAR CONSTANT
	DISPLAY_EST_RANGE_OFFSET	:	USINT	:=	10;
	DISPLAY_EST_RANGE_CF	:	USINT	:=	3;
	BATTERY_VOLTAGE_DISPLAY_CF	:	REAL	:=	0.25;
	DISPLAY_POWER_CF	:	UINT	:=	1000;
	DISPLAY_POWER_OFFSET	:	UINT	:=	32768;
	CHARGER_DETECTED	:	USINT	:=	0;
	
	
END_VAR


IF (gq_Gear_Neutral = TRUE) THEN
	gu16_CurrentGear	:=	0;
	gu16_CurrentGear1	:=	16#204E;
	gu8_CurrentGear2	:=	16#7D;
ELSIF (gq_Gear_Drive = TRUE) THEN
	gu16_CurrentGear	:=	16#2941;
	gu16_CurrentGear1	:=	16#2044;
	gu8_CurrentGear2	:=	16#7E;
ELSIF (gq_Gear_Reverse = TRUE) THEN
	gu16_CurrentGear	:=	16#2941;
	gu16_CurrentGear1	:=	16#2052;
	gu8_CurrentGear2	:=	16#7C;
END_IF

IF (Brusa1_Rx.StatusPP = CHARGER_DETECTED) THEN
	gq_CAN4_ChargerPP_Tx	:=	TRUE;
ELSE
	gq_CAN4_ChargerPP_Tx	:=	FALSE;
END_IF


(*601*)
gu16_CAN4_TripCounter_km_Tx			:=	00; (*0*)
gu16_CAN4_DisplayRangeMin_Tx		:=	00; (*0*)
gu16_CAN4_DisplayRangeMax_Tx		:=	00; (*0*)
gu16_CAN4_DisplayRangeEst_Tx		:=	LIMIT(0, (gu8_BMS_SOC - DISPLAY_EST_RANGE_OFFSET), 100) * DISPLAY_EST_RANGE_CF;
(*201*)
gs8_CAN4_CruiseControlSetpoint_Tx	:=	00; (*Need to add this when cruise control added*)
gs8_CAN4_DummyScreen601_Tx			:=	00; (*Need to find out what this is used for*)
gs8_CAN4_DisplayTemp_Tx				:=	INT_TO_SINT(gs16_MaxTemp_degC);
gs8_CAN4_DisplayDirection_Tx		:=	00; (*Bits*)
gs8_CAN4_DisplayDirection_Tx.4		:=	gq_Gear_Drive;
gs8_CAN4_DisplayDirection_Tx.5		:=	gq_Gear_Reverse;
gs8_CAN4_DisplayDirection_Tx.6		:=	gq_Gear_Neutral;
gs8_CAN4_DisplayDirection_Tx.7		:=	gq_HandBrake;
gs8_CAN4_SOC_Tx						:=	USINT_TO_SINT(gu8_BMS_SOC); (*SOC*)

gs8_CAN4_DisplayStatus_Tx.0		:=	00;
gs8_CAN4_DisplayStatus_Tx.1		:=	00;
gs8_CAN4_DisplayStatus_Tx.2		:=	gq_BMS1_AuxPosContactor; (*Aux Pos Cont 1*)
gs8_CAN4_DisplayStatus_Tx.3		:=	gq_BMS1_AuxNegContactor; (*Aux Neg Cont 1*)
gs8_CAN4_DisplayStatus_Tx.4		:=	gq_BMS2_AuxPosContactor; (*Aux Pos Cont 2*)
gs8_CAN4_DisplayStatus_Tx.5		:=	gq_BMS2_AuxNegContactor; (*Aux Neg Cont 2*)
gs8_CAN4_DisplayStatus_Tx.6		:=	gq_EStop; (*E Stop*)
gs8_CAN4_DisplayStatus_Tx.7		:=	gq_EStopLatch; (*E Stop Latch*)

gs8_CAN4_PowerIndicationRelative_Tx	:=	00; (*0*)
gs8_CAN4_DispVehicleStatus_Tx		:=	00; (*Bits, never set*)
(*301*)
gs8_CAN4_SOC1_Tx					:=	USINT_TO_SINT(gu8_BMS_SOC); (*SOC*)
gs8_CAN4_BatteryVoltage_Tx			:=	REAL_TO_SINT(gr_BMS_BatteryVoltage * BATTERY_VOLTAGE_DISPLAY_CF);
gs8_CAN4_MotorTemp_Tx				:=	REAL_TO_SINT(gr_MCU_ThermalIndicator); (*0*)
gs8_CAN4_InverterTemp_Tx			:=	REAL_TO_SINT(gr_MCU_ThermalIndicator); (*MCU Temp*)
gu8_CAN4_ChargerStatus_Tx.0			:=	00; (*0*)
gu8_CAN4_ChargerStatus_Tx.1			:=	00; (*0*)
gu8_CAN4_ChargerStatus_Tx.2			:=	00; (*0*)
gu8_CAN4_ChargerStatus_Tx.3			:=	gq_CAN4_ChargerPP_Tx; (*0*)
gu8_CAN4_ChargerStatus_Tx.4			:=	00; (*0*)
gu8_CAN4_ChargerStatus_Tx.5			:=	00; (*0*)
gu8_CAN4_ChargerStatus_Tx.6			:=	00; (*0*)
gu8_CAN4_ChargerStatus_Tx.7			:=	00; (*0*)
gs8_CAN4_ThrottlePedal_Tx			:=	REAL_TO_SINT(gr_AccelPedal_Perc * 100); (*Throttle Pedal*)
gs8_CAN4_BrakePedal_Tx				:=	00; (*0*)
gs8_CAN4_VehicleSpeedMsg_Tx			:=	00; (*0*)
(*401*)
gs8_CAN4_VehicleStatus_Tx			:=	00; (*Bits, never set*)
gs8_CAN4_VehicleStatus_Tx.1			:=	00; (*Door Open*)
gs8_CAN4_VehicleStatus_Tx.2			:=	00; (*Dashboard Illuminated*)
gs8_CAN4_VehicleStatus_Tx.3			:=	00; (*Power Steering*)
gs8_CAN4_VehicleStatus_Tx.4			:=	00; (*Air Compressor*)
gs8_CAN4_RegenTorquePercDisplay_Tx	:=	00; (*Scaled regen torque*)
gs16_CAN4_PowerIndication_Tx		:=	REAL_TO_INT((ABS(gr_BMS_BatteryVoltage * gs16_BMS_BatteryCurrent) / DISPLAY_POWER_CF) + DISPLAY_POWER_OFFSET); (*(current * batteryVoltage)*-1/1000)+32768*)
gs16_CAN4_BatteryCurrent_Tx			:=	gs16_BMS_BatteryCurrent; (*Current*)

IF (gu16_Sevcon1_Controlword = 5) THEN
	gq_Dash_Sevcon1_Enable	:=	TRUE;
ELSE
	gq_Dash_Sevcon1_Enable	:=	FALSE;
END_IF
IF (gu16_Sevcon2_Controlword = 5) THEN
	gq_Dash_Sevcon2_Enable	:=	TRUE;
ELSE
	gq_Dash_Sevcon2_Enable	:=	FALSE;
END_IF
IF (gu8_SystemState = DRIVE_SYS) THEN
	gq_Dash_Charge_Rq		:=	FALSE;
	gq_Dash_Discharge_Rq	:=	TRUE;
ELSIF (gu8_SystemState = PLUGIN_SYS) THEN
	gq_Dash_Charge_Rq		:=	TRUE;
	gq_Dash_Discharge_Rq	:=	FALSE;
ELSE
	gq_Dash_Charge_Rq		:=	FALSE;
	gq_Dash_Discharge_Rq	:=	FALSE;
END_IF
gs16_Dash_BattCurrent_Tx	:=	gs16_BMS_BatteryCurrent * 10;

IF (gu8_BMS_SOC >= 100 AND gs16_BMS1_CCL <= 0 AND gs16_BMS2_CCL <= 0) THEN
	gq_BattFullyCharged	:=	TRUE;
ELSE
	gq_BattFullyCharged	:=	FALSE;
END_IF

gu8_Dash_AccelPedal_Tx	:=	REAL_TO_USINT(gr_AccelPedal_Perc * 2.5);
gu8_Dash_BrakePressure1_Tx	:=	REAL_TO_USINT(gr_J1939_ServiceBrakeAirPressCircuit1 * 10);
gu8_Dash_BrakePressure2_Tx	:=	REAL_TO_USINT(gr_J1939_ServiceBrakeAirPressCircuit2 * 10);

gs16_Dash_Power	:=	REAL_TO_INT(gr_BMS_BatteryVoltage * gs16_BMS_BatteryCurrent * 0.001);

gs8_Dash_AverageTemp_Tx	:=	REAL_TO_SINT((gr_BMS_AverageTemp * 0.1) + 40);
gs8_Dash_HighTemp_Tx	:=	REAL_TO_SINT((gr_BMS_HighTemp * 0.1) + 40);
gs8_Dash_LowTemp_Tx	:=	REAL_TO_SINT((gr_BMS_LowTemp * 0.1) + 40);

gu8_BMS1_LowCellV_Tx	:=	UINT_TO_USINT(gu16_BMS1_LowCellVoltage / 1000);
gu8_BMS2_LowCellV_Tx	:=	UINT_TO_USINT(gu16_BMS2_LowCellVoltage / 1000);

END_PROGRAM

// Application/UserCode/CAN4/Data to or For HMI/BMS_to_HMI
PROGRAM BMS_to_HMI
VAR
	ht_CAN4_DD0_Tx	:	EPEC_CANVXD.Msg;
	ht_CAN4_DD1_Tx	:	EPEC_CANVXD.Msg;
	ht_CAN4_DD2_Tx	:	EPEC_CANVXD.Msg;
	ht_CAN4_DD3_Tx	:	EPEC_CANVXD.Msg;
	ht_CAN4_DD4_Tx	:	EPEC_CANVXD.Msg;
	ht_CAN4_DD5_Tx	:	EPEC_CANVXD.Msg;
	ht_CAN4_DD6_Tx	:	EPEC_CANVXD.Msg;
	ht_CAN4_DD7_Tx	:	EPEC_CANVXD.Msg;
	ht_CAN4_DD8_Tx	:	EPEC_CANVXD.Msg;
	ht_CAN4_DD9_Tx	:	EPEC_CANVXD.Msg;
	ht_CAN4_DDA_Tx	:	EPEC_CANVXD.Msg;
	ht_CAN4_DDB_Tx	:	EPEC_CANVXD.Msg;
	ht_CAN4_DDC_Tx	:	EPEC_CANVXD.Msg;
	ht_CAN4_DDD_Tx	:	EPEC_CANVXD.Msg;
	ht_CAN4_ADD0_Tx	:	EPEC_CANVXD.Msg;
	ht_CAN4_ADD1_Tx	:	EPEC_CANVXD.Msg;
	ht_CAN4_ADD2_Tx	:	EPEC_CANVXD.Msg;
	ht_CAN4_ADD3_Tx	:	EPEC_CANVXD.Msg;
	ht_CAN4_ADD4_Tx	:	EPEC_CANVXD.Msg;
	ht_CAN4_ADD5_Tx	:	EPEC_CANVXD.Msg;
	ht_CAN4_ADD6_Tx	:	EPEC_CANVXD.Msg;
	ht_CAN4_ADD7_Tx	:	EPEC_CANVXD.Msg;
	ht_CAN4_ADD8_Tx	:	EPEC_CANVXD.Msg;
	ht_CAN4_ADD9_Tx	:	EPEC_CANVXD.Msg;
	ht_CAN4_ADDA_Tx	:	EPEC_CANVXD.Msg;
	ht_CAN4_ADDB_Tx	:	EPEC_CANVXD.Msg;
	ht_CAN4_ADDC_Tx	:	EPEC_CANVXD.Msg;
	ht_CAN4_ADDD_Tx	:	EPEC_CANVXD.Msg;
	hton_MessageSend_Timer	:	TON;
	
	Tx_Timer	:	TON;
	
END_VAR

//Send raw BMS Data to HMI CAN#4
(*BMS1*)
ht_CAN4_DD0_Tx.ID		:=	16#181000DD OR EPEC_CANVXD.MASK_29BIT;
ht_CAN4_DD0_Tx.Data[0]	:=	OrionBMS1_Rx.OrionBMS1_6B0_Rx.au8_Data[0];
ht_CAN4_DD0_Tx.Data[1]	:=	OrionBMS1_Rx.OrionBMS1_6B0_Rx.au8_Data[1];
ht_CAN4_DD0_Tx.Data[2]	:=	OrionBMS1_Rx.OrionBMS1_6B0_Rx.au8_Data[2];
ht_CAN4_DD0_Tx.Data[3]	:=	OrionBMS1_Rx.OrionBMS1_6B0_Rx.au8_Data[3];
ht_CAN4_DD0_Tx.Data[4]	:=	OrionBMS1_Rx.OrionBMS1_6B0_Rx.au8_Data[4];
ht_CAN4_DD0_Tx.Data[5]	:=	OrionBMS1_Rx.OrionBMS1_6B0_Rx.au8_Data[5];		
ht_CAN4_DD0_Tx.Data[6]	:=	OrionBMS1_Rx.OrionBMS1_6B0_Rx.au8_Data[6];	
ht_CAN4_DD0_Tx.Data[7]	:=	OrionBMS1_Rx.OrionBMS1_6B0_Rx.au8_Data[7];		
ht_CAN4_DD0_Tx.Len		:=	8;

ht_CAN4_DD1_Tx.ID		:=	16#181001DD OR EPEC_CANVXD.MASK_29BIT;
ht_CAN4_DD1_Tx.Data[0]	:=	OrionBMS1_Rx.OrionBMS1_6B1_Rx.au8_Data[0];
ht_CAN4_DD1_Tx.Data[1]	:=	OrionBMS1_Rx.OrionBMS1_6B1_Rx.au8_Data[1];
ht_CAN4_DD1_Tx.Data[2]	:=	OrionBMS1_Rx.OrionBMS1_6B1_Rx.au8_Data[2];
ht_CAN4_DD1_Tx.Data[3]	:=	OrionBMS1_Rx.OrionBMS1_6B1_Rx.au8_Data[3];
ht_CAN4_DD1_Tx.Data[4]	:=	OrionBMS1_Rx.OrionBMS1_6B1_Rx.au8_Data[4];
ht_CAN4_DD1_Tx.Data[5]	:=	OrionBMS1_Rx.OrionBMS1_6B1_Rx.au8_Data[5];		
ht_CAN4_DD1_Tx.Data[6]	:=	OrionBMS1_Rx.OrionBMS1_6B1_Rx.au8_Data[6];	
ht_CAN4_DD1_Tx.Data[7]	:=	OrionBMS1_Rx.OrionBMS1_6B1_Rx.au8_Data[7];		
ht_CAN4_DD1_Tx.Len		:=	8;

ht_CAN4_DD2_Tx.ID		:=	16#181002DD OR EPEC_CANVXD.MASK_29BIT;
ht_CAN4_DD2_Tx.Data[0]	:=	OrionBMS1_Rx.OrionBMS1_6B2_Rx.au8_Data[0];
ht_CAN4_DD2_Tx.Data[1]	:=	OrionBMS1_Rx.OrionBMS1_6B2_Rx.au8_Data[1];
ht_CAN4_DD2_Tx.Data[2]	:=	OrionBMS1_Rx.OrionBMS1_6B2_Rx.au8_Data[2];
ht_CAN4_DD2_Tx.Data[3]	:=	OrionBMS1_Rx.OrionBMS1_6B2_Rx.au8_Data[3];
ht_CAN4_DD2_Tx.Data[4]	:=	OrionBMS1_Rx.OrionBMS1_6B2_Rx.au8_Data[4];
ht_CAN4_DD2_Tx.Data[5]	:=	OrionBMS1_Rx.OrionBMS1_6B2_Rx.au8_Data[5];		
ht_CAN4_DD2_Tx.Data[6]	:=	OrionBMS1_Rx.OrionBMS1_6B2_Rx.au8_Data[6];	
ht_CAN4_DD2_Tx.Data[7]	:=	OrionBMS1_Rx.OrionBMS1_6B2_Rx.au8_Data[7];		
ht_CAN4_DD2_Tx.Len		:=	8;

ht_CAN4_DD3_Tx.ID		:=	16#181003DD OR EPEC_CANVXD.MASK_29BIT;
ht_CAN4_DD3_Tx.Data[0]	:=	OrionBMS1_Rx.OrionBMS1_6B3_Rx.au8_Data[0];
ht_CAN4_DD3_Tx.Data[1]	:=	OrionBMS1_Rx.OrionBMS1_6B3_Rx.au8_Data[1];
ht_CAN4_DD3_Tx.Data[2]	:=	OrionBMS1_Rx.OrionBMS1_6B3_Rx.au8_Data[2];
ht_CAN4_DD3_Tx.Data[3]	:=	OrionBMS1_Rx.OrionBMS1_6B3_Rx.au8_Data[3];
ht_CAN4_DD3_Tx.Data[4]	:=	OrionBMS1_Rx.OrionBMS1_6B3_Rx.au8_Data[4];
ht_CAN4_DD3_Tx.Data[5]	:=	OrionBMS1_Rx.OrionBMS1_6B3_Rx.au8_Data[5];		
ht_CAN4_DD3_Tx.Data[6]	:=	OrionBMS1_Rx.OrionBMS1_6B3_Rx.au8_Data[6];	
ht_CAN4_DD3_Tx.Data[7]	:=	OrionBMS1_Rx.OrionBMS1_6B3_Rx.au8_Data[7];		
ht_CAN4_DD3_Tx.Len		:=	8;

ht_CAN4_DD4_Tx.ID		:=	16#181004DD OR EPEC_CANVXD.MASK_29BIT;
ht_CAN4_DD4_Tx.Data[0]	:=	OrionBMS1_Rx.OrionBMS1_6B4_Rx.au8_Data[0];
ht_CAN4_DD4_Tx.Data[1]	:=	OrionBMS1_Rx.OrionBMS1_6B4_Rx.au8_Data[1];
ht_CAN4_DD4_Tx.Data[2]	:=	OrionBMS1_Rx.OrionBMS1_6B4_Rx.au8_Data[2];
ht_CAN4_DD4_Tx.Data[3]	:=	OrionBMS1_Rx.OrionBMS1_6B4_Rx.au8_Data[3];
ht_CAN4_DD4_Tx.Data[4]	:=	OrionBMS1_Rx.OrionBMS1_6B4_Rx.au8_Data[4];
ht_CAN4_DD4_Tx.Data[5]	:=	OrionBMS1_Rx.OrionBMS1_6B4_Rx.au8_Data[5];		
ht_CAN4_DD4_Tx.Data[6]	:=	OrionBMS1_Rx.OrionBMS1_6B4_Rx.au8_Data[6];	
ht_CAN4_DD4_Tx.Data[7]	:=	OrionBMS1_Rx.OrionBMS1_6B4_Rx.au8_Data[7];		
ht_CAN4_DD4_Tx.Len		:=	8;

ht_CAN4_DD5_Tx.ID		:=	16#181005DD OR EPEC_CANVXD.MASK_29BIT;
ht_CAN4_DD5_Tx.Data[0]	:=	OrionBMS1_Rx.OrionBMS1_6B5_Rx.au8_Data[0];
ht_CAN4_DD5_Tx.Data[1]	:=	OrionBMS1_Rx.OrionBMS1_6B5_Rx.au8_Data[1];
ht_CAN4_DD5_Tx.Data[2]	:=	OrionBMS1_Rx.OrionBMS1_6B5_Rx.au8_Data[2];
ht_CAN4_DD5_Tx.Data[3]	:=	OrionBMS1_Rx.OrionBMS1_6B5_Rx.au8_Data[3];
ht_CAN4_DD5_Tx.Data[4]	:=	OrionBMS1_Rx.OrionBMS1_6B5_Rx.au8_Data[4];
ht_CAN4_DD5_Tx.Data[5]	:=	OrionBMS1_Rx.OrionBMS1_6B5_Rx.au8_Data[5];		
ht_CAN4_DD5_Tx.Data[6]	:=	OrionBMS1_Rx.OrionBMS1_6B5_Rx.au8_Data[6];	
ht_CAN4_DD5_Tx.Data[7]	:=	OrionBMS1_Rx.OrionBMS1_6B5_Rx.au8_Data[7];		
ht_CAN4_DD5_Tx.Len		:=	8;

ht_CAN4_DD6_Tx.ID		:=	16#181006DD OR EPEC_CANVXD.MASK_29BIT;
ht_CAN4_DD6_Tx.Data[0]	:=	OrionBMS1_Rx.OrionBMS1_6B6_Rx.au8_Data[0];
ht_CAN4_DD6_Tx.Data[1]	:=	OrionBMS1_Rx.OrionBMS1_6B6_Rx.au8_Data[1];
ht_CAN4_DD6_Tx.Data[2]	:=	OrionBMS1_Rx.OrionBMS1_6B6_Rx.au8_Data[2];
ht_CAN4_DD6_Tx.Data[3]	:=	OrionBMS1_Rx.OrionBMS1_6B6_Rx.au8_Data[3];
ht_CAN4_DD6_Tx.Data[4]	:=	OrionBMS1_Rx.OrionBMS1_6B6_Rx.au8_Data[4];
ht_CAN4_DD6_Tx.Data[5]	:=	OrionBMS1_Rx.OrionBMS1_6B6_Rx.au8_Data[5];		
ht_CAN4_DD6_Tx.Data[6]	:=	OrionBMS1_Rx.OrionBMS1_6B6_Rx.au8_Data[6];	
ht_CAN4_DD6_Tx.Data[7]	:=	OrionBMS1_Rx.OrionBMS1_6B6_Rx.au8_Data[7];		
ht_CAN4_DD6_Tx.Len		:=	8;

ht_CAN4_DD7_Tx.ID		:=	16#181007DD OR EPEC_CANVXD.MASK_29BIT;
ht_CAN4_DD7_Tx.Data[0]	:=	OrionBMS1_Rx.OrionBMS1_6B7_Rx.au8_Data[0];
ht_CAN4_DD7_Tx.Data[1]	:=	OrionBMS1_Rx.OrionBMS1_6B7_Rx.au8_Data[1];
ht_CAN4_DD7_Tx.Data[2]	:=	OrionBMS1_Rx.OrionBMS1_6B7_Rx.au8_Data[2];
ht_CAN4_DD7_Tx.Data[3]	:=	OrionBMS1_Rx.OrionBMS1_6B7_Rx.au8_Data[3];
ht_CAN4_DD7_Tx.Data[4]	:=	OrionBMS1_Rx.OrionBMS1_6B7_Rx.au8_Data[4];
ht_CAN4_DD7_Tx.Data[5]	:=	OrionBMS1_Rx.OrionBMS1_6B7_Rx.au8_Data[5];		
ht_CAN4_DD7_Tx.Data[6]	:=	OrionBMS1_Rx.OrionBMS1_6B7_Rx.au8_Data[6];	
ht_CAN4_DD7_Tx.Data[7]	:=	OrionBMS1_Rx.OrionBMS1_6B7_Rx.au8_Data[7];		
ht_CAN4_DD7_Tx.Len		:=	8;

ht_CAN4_DD8_Tx.ID		:=	16#181008DD OR EPEC_CANVXD.MASK_29BIT;
ht_CAN4_DD8_Tx.Data[0]	:=	OrionBMS1_Rx.OrionBMS1_6B8_Rx.au8_Data[0];
ht_CAN4_DD8_Tx.Data[1]	:=	OrionBMS1_Rx.OrionBMS1_6B8_Rx.au8_Data[1];
ht_CAN4_DD8_Tx.Data[2]	:=	OrionBMS1_Rx.OrionBMS1_6B8_Rx.au8_Data[2];
ht_CAN4_DD8_Tx.Data[3]	:=	OrionBMS1_Rx.OrionBMS1_6B8_Rx.au8_Data[3];
ht_CAN4_DD8_Tx.Data[4]	:=	OrionBMS1_Rx.OrionBMS1_6B8_Rx.au8_Data[4];
ht_CAN4_DD8_Tx.Data[5]	:=	OrionBMS1_Rx.OrionBMS1_6B8_Rx.au8_Data[5];		
ht_CAN4_DD8_Tx.Data[6]	:=	OrionBMS1_Rx.OrionBMS1_6B8_Rx.au8_Data[6];	
ht_CAN4_DD8_Tx.Data[7]	:=	OrionBMS1_Rx.OrionBMS1_6B8_Rx.au8_Data[7];		
ht_CAN4_DD8_Tx.Len		:=	8;

ht_CAN4_DD9_Tx.ID		:=	16#181009DD OR EPEC_CANVXD.MASK_29BIT;
ht_CAN4_DD9_Tx.Data[0]	:=	OrionBMS1_Rx.OrionBMS1_6B9_Rx.au8_Data[0];
ht_CAN4_DD9_Tx.Data[1]	:=	OrionBMS1_Rx.OrionBMS1_6B9_Rx.au8_Data[1];
ht_CAN4_DD9_Tx.Data[2]	:=	OrionBMS1_Rx.OrionBMS1_6B9_Rx.au8_Data[2];
ht_CAN4_DD9_Tx.Data[3]	:=	OrionBMS1_Rx.OrionBMS1_6B9_Rx.au8_Data[3];
ht_CAN4_DD9_Tx.Data[4]	:=	OrionBMS1_Rx.OrionBMS1_6B9_Rx.au8_Data[4];
ht_CAN4_DD9_Tx.Data[5]	:=	OrionBMS1_Rx.OrionBMS1_6B9_Rx.au8_Data[5];		
ht_CAN4_DD9_Tx.Data[6]	:=	OrionBMS1_Rx.OrionBMS1_6B9_Rx.au8_Data[6];	
ht_CAN4_DD9_Tx.Data[7]	:=	OrionBMS1_Rx.OrionBMS1_6B9_Rx.au8_Data[7];		
ht_CAN4_DD9_Tx.Len		:=	8;

ht_CAN4_DDA_Tx.ID		:=	16#18100ADD OR EPEC_CANVXD.MASK_29BIT;
ht_CAN4_DDA_Tx.Data[0]	:=	OrionBMS1_Rx.OrionBMS1_6BA_Rx.au8_Data[0];
ht_CAN4_DDA_Tx.Data[1]	:=	OrionBMS1_Rx.OrionBMS1_6BA_Rx.au8_Data[1];
ht_CAN4_DDA_Tx.Data[2]	:=	OrionBMS1_Rx.OrionBMS1_6BA_Rx.au8_Data[2];
ht_CAN4_DDA_Tx.Data[3]	:=	OrionBMS1_Rx.OrionBMS1_6BA_Rx.au8_Data[3];
ht_CAN4_DDA_Tx.Data[4]	:=	OrionBMS1_Rx.OrionBMS1_6BA_Rx.au8_Data[4];
ht_CAN4_DDA_Tx.Data[5]	:=	OrionBMS1_Rx.OrionBMS1_6BA_Rx.au8_Data[5];		
ht_CAN4_DDA_Tx.Data[6]	:=	OrionBMS1_Rx.OrionBMS1_6BA_Rx.au8_Data[6];	
ht_CAN4_DDA_Tx.Data[7]	:=	OrionBMS1_Rx.OrionBMS1_6BA_Rx.au8_Data[7];		
ht_CAN4_DDA_Tx.Len		:=	8;

ht_CAN4_DDB_Tx.ID		:=	16#18100BDD OR EPEC_CANVXD.MASK_29BIT;
ht_CAN4_DDB_Tx.Data[0]	:=	OrionBMS1_Rx.OrionBMS1_6BB_Rx.au8_Data[0];
ht_CAN4_DDB_Tx.Data[1]	:=	OrionBMS1_Rx.OrionBMS1_6BB_Rx.au8_Data[1];
ht_CAN4_DDB_Tx.Data[2]	:=	OrionBMS1_Rx.OrionBMS1_6BB_Rx.au8_Data[2];
ht_CAN4_DDB_Tx.Data[3]	:=	OrionBMS1_Rx.OrionBMS1_6BB_Rx.au8_Data[3];
ht_CAN4_DDB_Tx.Data[4]	:=	OrionBMS1_Rx.OrionBMS1_6BB_Rx.au8_Data[4];
ht_CAN4_DDB_Tx.Data[5]	:=	OrionBMS1_Rx.OrionBMS1_6BB_Rx.au8_Data[5];		
ht_CAN4_DDB_Tx.Data[6]	:=	OrionBMS1_Rx.OrionBMS1_6BB_Rx.au8_Data[6];	
ht_CAN4_DDB_Tx.Data[7]	:=	OrionBMS1_Rx.OrionBMS1_6BB_Rx.au8_Data[7];		
ht_CAN4_DDB_Tx.Len		:=	8;

ht_CAN4_DDC_Tx.ID		:=	16#18100CDD OR EPEC_CANVXD.MASK_29BIT;
ht_CAN4_DDC_Tx.Data[0]	:=	OrionBMS1_Rx.OrionBMS1_6BC_Rx.au8_Data[0];
ht_CAN4_DDC_Tx.Data[1]	:=	OrionBMS1_Rx.OrionBMS1_6BC_Rx.au8_Data[1];
ht_CAN4_DDC_Tx.Data[2]	:=	OrionBMS1_Rx.OrionBMS1_6BC_Rx.au8_Data[2];
ht_CAN4_DDC_Tx.Data[3]	:=	OrionBMS1_Rx.OrionBMS1_6BC_Rx.au8_Data[3];
ht_CAN4_DDC_Tx.Data[4]	:=	OrionBMS1_Rx.OrionBMS1_6BC_Rx.au8_Data[4];
ht_CAN4_DDC_Tx.Data[5]	:=	OrionBMS1_Rx.OrionBMS1_6BC_Rx.au8_Data[5];		
ht_CAN4_DDC_Tx.Data[6]	:=	OrionBMS1_Rx.OrionBMS1_6BC_Rx.au8_Data[6];	
ht_CAN4_DDC_Tx.Data[7]	:=	OrionBMS1_Rx.OrionBMS1_6BC_Rx.au8_Data[7];		
ht_CAN4_DDC_Tx.Len		:=	8;

ht_CAN4_DDD_Tx.ID		:=	16#18100DDD OR EPEC_CANVXD.MASK_29BIT;
ht_CAN4_DDD_Tx.Data[0]	:=	OrionBMS1_Rx.OrionBMS1_6BD_Rx.au8_Data[0];
ht_CAN4_DDD_Tx.Data[1]	:=	OrionBMS1_Rx.OrionBMS1_6BD_Rx.au8_Data[1];
ht_CAN4_DDD_Tx.Data[2]	:=	OrionBMS1_Rx.OrionBMS1_6BD_Rx.au8_Data[2];
ht_CAN4_DDD_Tx.Data[3]	:=	OrionBMS1_Rx.OrionBMS1_6BD_Rx.au8_Data[3];
ht_CAN4_DDD_Tx.Data[4]	:=	OrionBMS1_Rx.OrionBMS1_6BD_Rx.au8_Data[4];
ht_CAN4_DDD_Tx.Data[5]	:=	OrionBMS1_Rx.OrionBMS1_6BD_Rx.au8_Data[5];		
ht_CAN4_DDD_Tx.Data[6]	:=	OrionBMS1_Rx.OrionBMS1_6BD_Rx.au8_Data[6];	
ht_CAN4_DDD_Tx.Data[7]	:=	OrionBMS1_Rx.OrionBMS1_6BD_Rx.au8_Data[7];		
ht_CAN4_DDD_Tx.Len		:=	8;

//*BMS Slave
ht_CAN4_ADD0_Tx.ID		:=	16#182000DD OR EPEC_CANVXD.MASK_29BIT;
ht_CAN4_ADD0_Tx.Data[0]	:=	OrionBMS2_Rx.OrionBMS2_6B0_Rx.au8_Data[0];
ht_CAN4_ADD0_Tx.Data[1]	:=	OrionBMS2_Rx.OrionBMS2_6B0_Rx.au8_Data[1];
ht_CAN4_ADD0_Tx.Data[2]	:=	OrionBMS2_Rx.OrionBMS2_6B0_Rx.au8_Data[2];
ht_CAN4_ADD0_Tx.Data[3]	:=	OrionBMS2_Rx.OrionBMS2_6B0_Rx.au8_Data[3];
ht_CAN4_ADD0_Tx.Data[4]	:=	OrionBMS2_Rx.OrionBMS2_6B0_Rx.au8_Data[4];
ht_CAN4_ADD0_Tx.Data[5]	:=	OrionBMS2_Rx.OrionBMS2_6B0_Rx.au8_Data[5];		
ht_CAN4_ADD0_Tx.Data[6]	:=	OrionBMS2_Rx.OrionBMS2_6B0_Rx.au8_Data[6];	
ht_CAN4_ADD0_Tx.Data[7]	:=	OrionBMS2_Rx.OrionBMS2_6B0_Rx.au8_Data[7];		
ht_CAN4_ADD0_Tx.Len		:=	8;

ht_CAN4_ADD1_Tx.ID		:=	16#182001DD OR EPEC_CANVXD.MASK_29BIT;
ht_CAN4_ADD1_Tx.Data[0]	:=	OrionBMS2_Rx.OrionBMS2_6B1_Rx.au8_Data[0];
ht_CAN4_ADD1_Tx.Data[1]	:=	OrionBMS2_Rx.OrionBMS2_6B1_Rx.au8_Data[1];
ht_CAN4_ADD1_Tx.Data[2]	:=	OrionBMS2_Rx.OrionBMS2_6B1_Rx.au8_Data[2];
ht_CAN4_ADD1_Tx.Data[3]	:=	OrionBMS2_Rx.OrionBMS2_6B1_Rx.au8_Data[3];
ht_CAN4_ADD1_Tx.Data[4]	:=	OrionBMS2_Rx.OrionBMS2_6B1_Rx.au8_Data[4];
ht_CAN4_ADD1_Tx.Data[5]	:=	OrionBMS2_Rx.OrionBMS2_6B1_Rx.au8_Data[5];		
ht_CAN4_ADD1_Tx.Data[6]	:=	OrionBMS2_Rx.OrionBMS2_6B1_Rx.au8_Data[6];	
ht_CAN4_ADD1_Tx.Data[7]	:=	OrionBMS2_Rx.OrionBMS2_6B1_Rx.au8_Data[7];		
ht_CAN4_ADD1_Tx.Len		:=	8;

ht_CAN4_ADD2_Tx.ID		:=	16#182002DD OR EPEC_CANVXD.MASK_29BIT;
ht_CAN4_ADD2_Tx.Data[0]	:=	OrionBMS2_Rx.OrionBMS2_6B2_Rx.au8_Data[0];
ht_CAN4_ADD2_Tx.Data[1]	:=	OrionBMS2_Rx.OrionBMS2_6B2_Rx.au8_Data[1];
ht_CAN4_ADD2_Tx.Data[2]	:=	OrionBMS2_Rx.OrionBMS2_6B2_Rx.au8_Data[2];
ht_CAN4_ADD2_Tx.Data[3]	:=	OrionBMS2_Rx.OrionBMS2_6B2_Rx.au8_Data[3];
ht_CAN4_ADD2_Tx.Data[4]	:=	OrionBMS2_Rx.OrionBMS2_6B2_Rx.au8_Data[4];
ht_CAN4_ADD2_Tx.Data[5]	:=	OrionBMS2_Rx.OrionBMS2_6B2_Rx.au8_Data[5];		
ht_CAN4_ADD2_Tx.Data[6]	:=	OrionBMS2_Rx.OrionBMS2_6B2_Rx.au8_Data[6];	
ht_CAN4_ADD2_Tx.Data[7]	:=	OrionBMS2_Rx.OrionBMS2_6B2_Rx.au8_Data[7];		
ht_CAN4_ADD2_Tx.Len		:=	8;

ht_CAN4_ADD3_Tx.ID		:=	16#182003DD OR EPEC_CANVXD.MASK_29BIT;
ht_CAN4_ADD3_Tx.Data[0]	:=	OrionBMS2_Rx.OrionBMS2_6B3_Rx.au8_Data[0];
ht_CAN4_ADD3_Tx.Data[1]	:=	OrionBMS2_Rx.OrionBMS2_6B3_Rx.au8_Data[1];
ht_CAN4_ADD3_Tx.Data[2]	:=	OrionBMS2_Rx.OrionBMS2_6B3_Rx.au8_Data[2];
ht_CAN4_ADD3_Tx.Data[3]	:=	OrionBMS2_Rx.OrionBMS2_6B3_Rx.au8_Data[3];
ht_CAN4_ADD3_Tx.Data[4]	:=	OrionBMS2_Rx.OrionBMS2_6B3_Rx.au8_Data[4];
ht_CAN4_ADD3_Tx.Data[5]	:=	OrionBMS2_Rx.OrionBMS2_6B3_Rx.au8_Data[5];		
ht_CAN4_ADD3_Tx.Data[6]	:=	OrionBMS2_Rx.OrionBMS2_6B3_Rx.au8_Data[6];	
ht_CAN4_ADD3_Tx.Data[7]	:=	OrionBMS2_Rx.OrionBMS2_6B3_Rx.au8_Data[7];		
ht_CAN4_ADD3_Tx.Len		:=	8;

ht_CAN4_ADD4_Tx.ID		:=	16#182004DD OR EPEC_CANVXD.MASK_29BIT;
ht_CAN4_ADD4_Tx.Data[0]	:=	OrionBMS2_Rx.OrionBMS2_6B4_Rx.au8_Data[0];
ht_CAN4_ADD4_Tx.Data[1]	:=	OrionBMS2_Rx.OrionBMS2_6B4_Rx.au8_Data[1];
ht_CAN4_ADD4_Tx.Data[2]	:=	OrionBMS2_Rx.OrionBMS2_6B4_Rx.au8_Data[2];
ht_CAN4_ADD4_Tx.Data[3]	:=	OrionBMS2_Rx.OrionBMS2_6B4_Rx.au8_Data[3];
ht_CAN4_ADD4_Tx.Data[4]	:=	OrionBMS2_Rx.OrionBMS2_6B4_Rx.au8_Data[4];
ht_CAN4_ADD4_Tx.Data[5]	:=	OrionBMS2_Rx.OrionBMS2_6B4_Rx.au8_Data[5];		
ht_CAN4_ADD4_Tx.Data[6]	:=	OrionBMS2_Rx.OrionBMS2_6B4_Rx.au8_Data[6];	
ht_CAN4_ADD4_Tx.Data[7]	:=	OrionBMS2_Rx.OrionBMS2_6B4_Rx.au8_Data[7];		
ht_CAN4_ADD4_Tx.Len		:=	8;

ht_CAN4_ADD5_Tx.ID		:=	16#182005DD OR EPEC_CANVXD.MASK_29BIT;
ht_CAN4_ADD5_Tx.Data[0]	:=	OrionBMS2_Rx.OrionBMS2_6B5_Rx.au8_Data[0];
ht_CAN4_ADD5_Tx.Data[1]	:=	OrionBMS2_Rx.OrionBMS2_6B5_Rx.au8_Data[1];
ht_CAN4_ADD5_Tx.Data[2]	:=	OrionBMS2_Rx.OrionBMS2_6B5_Rx.au8_Data[2];
ht_CAN4_ADD5_Tx.Data[3]	:=	OrionBMS2_Rx.OrionBMS2_6B5_Rx.au8_Data[3];
ht_CAN4_ADD5_Tx.Data[4]	:=	OrionBMS2_Rx.OrionBMS2_6B5_Rx.au8_Data[4];
ht_CAN4_ADD5_Tx.Data[5]	:=	OrionBMS2_Rx.OrionBMS2_6B5_Rx.au8_Data[5];		
ht_CAN4_ADD5_Tx.Data[6]	:=	OrionBMS2_Rx.OrionBMS2_6B5_Rx.au8_Data[6];	
ht_CAN4_ADD5_Tx.Data[7]	:=	OrionBMS2_Rx.OrionBMS2_6B5_Rx.au8_Data[7];		
ht_CAN4_ADD5_Tx.Len		:=	8;

ht_CAN4_ADD6_Tx.ID		:=	16#182006DD OR EPEC_CANVXD.MASK_29BIT;
ht_CAN4_ADD6_Tx.Data[0]	:=	OrionBMS2_Rx.OrionBMS2_6B6_Rx.au8_Data[0];
ht_CAN4_ADD6_Tx.Data[1]	:=	OrionBMS2_Rx.OrionBMS2_6B6_Rx.au8_Data[1];
ht_CAN4_ADD6_Tx.Data[2]	:=	OrionBMS2_Rx.OrionBMS2_6B6_Rx.au8_Data[2];
ht_CAN4_ADD6_Tx.Data[3]	:=	OrionBMS2_Rx.OrionBMS2_6B6_Rx.au8_Data[3];
ht_CAN4_ADD6_Tx.Data[4]	:=	OrionBMS2_Rx.OrionBMS2_6B6_Rx.au8_Data[4];
ht_CAN4_ADD6_Tx.Data[5]	:=	OrionBMS2_Rx.OrionBMS2_6B6_Rx.au8_Data[5];		
ht_CAN4_ADD6_Tx.Data[6]	:=	OrionBMS2_Rx.OrionBMS2_6B6_Rx.au8_Data[6];	
ht_CAN4_ADD6_Tx.Data[7]	:=	OrionBMS2_Rx.OrionBMS2_6B6_Rx.au8_Data[7];		
ht_CAN4_ADD6_Tx.Len		:=	8;

ht_CAN4_ADD7_Tx.ID		:=	16#182007DD OR EPEC_CANVXD.MASK_29BIT;
ht_CAN4_ADD7_Tx.Data[0]	:=	OrionBMS2_Rx.OrionBMS2_6B7_Rx.au8_Data[0];
ht_CAN4_ADD7_Tx.Data[1]	:=	OrionBMS2_Rx.OrionBMS2_6B7_Rx.au8_Data[1];
ht_CAN4_ADD7_Tx.Data[2]	:=	OrionBMS2_Rx.OrionBMS2_6B7_Rx.au8_Data[2];
ht_CAN4_ADD7_Tx.Data[3]	:=	OrionBMS2_Rx.OrionBMS2_6B7_Rx.au8_Data[3];
ht_CAN4_ADD7_Tx.Data[4]	:=	OrionBMS2_Rx.OrionBMS2_6B7_Rx.au8_Data[4];
ht_CAN4_ADD7_Tx.Data[5]	:=	OrionBMS2_Rx.OrionBMS2_6B7_Rx.au8_Data[5];		
ht_CAN4_ADD7_Tx.Data[6]	:=	OrionBMS2_Rx.OrionBMS2_6B7_Rx.au8_Data[6];	
ht_CAN4_ADD7_Tx.Data[7]	:=	OrionBMS2_Rx.OrionBMS2_6B7_Rx.au8_Data[7];		
ht_CAN4_ADD7_Tx.Len		:=	8;

ht_CAN4_ADD8_Tx.ID		:=	16#182008DD OR EPEC_CANVXD.MASK_29BIT;
ht_CAN4_ADD8_Tx.Data[0]	:=	OrionBMS2_Rx.OrionBMS2_6B8_Rx.au8_Data[0];
ht_CAN4_ADD8_Tx.Data[1]	:=	OrionBMS2_Rx.OrionBMS2_6B8_Rx.au8_Data[1];
ht_CAN4_ADD8_Tx.Data[2]	:=	OrionBMS2_Rx.OrionBMS2_6B8_Rx.au8_Data[2];
ht_CAN4_ADD8_Tx.Data[3]	:=	OrionBMS2_Rx.OrionBMS2_6B8_Rx.au8_Data[3];
ht_CAN4_ADD8_Tx.Data[4]	:=	OrionBMS2_Rx.OrionBMS2_6B8_Rx.au8_Data[4];
ht_CAN4_ADD8_Tx.Data[5]	:=	OrionBMS2_Rx.OrionBMS2_6B8_Rx.au8_Data[5];		
ht_CAN4_ADD8_Tx.Data[6]	:=	OrionBMS2_Rx.OrionBMS2_6B8_Rx.au8_Data[6];	
ht_CAN4_ADD8_Tx.Data[7]	:=	OrionBMS2_Rx.OrionBMS2_6B8_Rx.au8_Data[7];		
ht_CAN4_ADD8_Tx.Len		:=	8;

ht_CAN4_ADD9_Tx.ID		:=	16#182009DD OR EPEC_CANVXD.MASK_29BIT;
ht_CAN4_ADD9_Tx.Data[0]	:=	OrionBMS2_Rx.OrionBMS2_6B9_Rx.au8_Data[0];
ht_CAN4_ADD9_Tx.Data[1]	:=	OrionBMS2_Rx.OrionBMS2_6B9_Rx.au8_Data[1];
ht_CAN4_ADD9_Tx.Data[2]	:=	OrionBMS2_Rx.OrionBMS2_6B9_Rx.au8_Data[2];
ht_CAN4_ADD9_Tx.Data[3]	:=	OrionBMS2_Rx.OrionBMS2_6B9_Rx.au8_Data[3];
ht_CAN4_ADD9_Tx.Data[4]	:=	OrionBMS2_Rx.OrionBMS2_6B9_Rx.au8_Data[4];
ht_CAN4_ADD9_Tx.Data[5]	:=	OrionBMS2_Rx.OrionBMS2_6B9_Rx.au8_Data[5];		
ht_CAN4_ADD9_Tx.Data[6]	:=	OrionBMS2_Rx.OrionBMS2_6B9_Rx.au8_Data[6];	
ht_CAN4_ADD9_Tx.Data[7]	:=	OrionBMS2_Rx.OrionBMS2_6B9_Rx.au8_Data[7];		
ht_CAN4_ADD9_Tx.Len		:=	8;

ht_CAN4_ADDA_Tx.ID		:=	16#18200ADD OR EPEC_CANVXD.MASK_29BIT;
ht_CAN4_ADDA_Tx.Data[0]	:=	OrionBMS2_Rx.OrionBMS2_6BA_Rx.au8_Data[0];
ht_CAN4_ADDA_Tx.Data[1]	:=	OrionBMS2_Rx.OrionBMS2_6BA_Rx.au8_Data[1];
ht_CAN4_ADDA_Tx.Data[2]	:=	OrionBMS2_Rx.OrionBMS2_6BA_Rx.au8_Data[2];
ht_CAN4_ADDA_Tx.Data[3]	:=	OrionBMS2_Rx.OrionBMS2_6BA_Rx.au8_Data[3];
ht_CAN4_ADDA_Tx.Data[4]	:=	OrionBMS2_Rx.OrionBMS2_6BA_Rx.au8_Data[4];
ht_CAN4_ADDA_Tx.Data[5]	:=	OrionBMS2_Rx.OrionBMS2_6BA_Rx.au8_Data[5];		
ht_CAN4_ADDA_Tx.Data[6]	:=	OrionBMS2_Rx.OrionBMS2_6BA_Rx.au8_Data[6];	
ht_CAN4_ADDA_Tx.Data[7]	:=	OrionBMS2_Rx.OrionBMS2_6BA_Rx.au8_Data[7];		
ht_CAN4_ADDA_Tx.Len		:=	8;

